LIN {X 0,Y 525.784,Z 203.51,A -85,B 0,C 180,E1 -4784.972,E2 -4784.972} C_VEL
LIN {X 0,Y 524.23,Z 193.259,A -85,B 0,C 180,E1 -4785.175,E2 -4785.175} C_VEL
LIN {X 0,Y 524.605,Z 174.888,A -85,B 0,C 180,E1 -4787.978,E2 -4787.978} C_VEL
LIN {X 0,Y 525.075,Z 155.446,A -85,B 0,C 180,E1 -4790.98,E2 -4790.98} C_VEL
LIN {X 0,Y 525.35,Z 141.019,A -85,B 0,C 180,E1 -4793.244,E2 -4793.244} C_VEL
LIN {X 0,Y 523.931,Z 133.223,A -85,B 0,C 180,E1 -4794.572,E2 -4794.572} C_VEL
LIN {X 0,Y 523.922,Z 133.227,A -85,B 0,C 180,E1 -4797.706,E2 -4797.706} C_VEL
LIN {X 0,Y 523.948,Z 133.217,A -85,B 0,C 180,E1 -4800.645,E2 -4800.645} C_VEL
LIN {X 0,Y 523.93,Z 133.224,A -85,B 0,C 180,E1 -4803.729,E2 -4803.729} C_VEL
LIN {X 0,Y 523.902,Z 133.221,A -85,B 0,C 180,E1 -4806.4,E2 -4806.4} C_VEL
LIN {X 0,Y 523.916,Z 133.222,A -85,B 0,C 180,E1 -4809.086,E2 -4809.086} C_VEL
LIN {X 0,Y 523.903,Z 133.221,A -85,B 0,C 180,E1 -4812.124,E2 -4812.124} C_VEL
LIN {X 0,Y 523.938,Z 133.225,A -85,B 0,C 180,E1 -4815.311,E2 -4815.311} C_VEL
LIN {X 0,Y 523.925,Z 133.22,A -85,B 0,C 180,E1 -4818.694,E2 -4818.694} C_VEL
LIN {X 0,Y 523.916,Z 133.219,A -85,B 0,C 180,E1 -4821.898,E2 -4821.898} C_VEL
LIN {X 0,Y 523.922,Z 133.225,A -85,B 0,C 180,E1 -4824.912,E2 -4824.912} C_VEL
LIN {X 0,Y 523.935,Z 133.217,A -85,B 0,C 180,E1 -4827.681,E2 -4827.681} C_VEL
LIN {X 0,Y 523.936,Z 133.221,A -85,B 0,C 180,E1 -4830.681,E2 -4830.681} C_VEL
LIN {X 0,Y 523.908,Z 133.22,A -85,B 0,C 180,E1 -4833.724,E2 -4833.724} C_VEL
LIN {X 0,Y 523.903,Z 133.222,A -85,B 0,C 180,E1 -4836.269,E2 -4836.269} C_VEL
LIN {X 0,Y 523.929,Z 133.226,A -85,B 0,C 180,E1 -4838.765,E2 -4838.765} C_VEL
LIN {X 0,Y 523.931,Z 133.219,A -85,B 0,C 180,E1 -4841.219,E2 -4841.219} C_VEL
LIN {X 0,Y 523.915,Z 133.225,A -85,B 0,C 180,E1 -4844.437,E2 -4844.437} C_VEL
LIN {X 0,Y 523.955,Z 133.214,A -85,B 0,C 180,E1 -4847.607,E2 -4847.607} C_VEL
LIN {X 0,Y 523.933,Z 133.219,A -85,B 0,C 180,E1 -4849.957,E2 -4849.957} C_VEL
LIN {X 0,Y 523.997,Z 133.209,A -85,B 0,C 180,E1 -4853.066,E2 -4853.066} C_VEL
LIN {X 0,Y 523.95,Z 133.214,A -85,B 0,C 180,E1 -4855.383,E2 -4855.383} C_VEL
LIN {X 0,Y 524.107,Z 133.196,A -85,B 0,C 180,E1 -4857.694,E2 -4857.694} C_VEL
LIN {X 0,Y 524.1,Z 133.201,A -85,B 0,C 180,E1 -4859.999,E2 -4859.999} C_VEL
LIN {X 0,Y 524.107,Z 133.202,A -85,B 0,C 180,E1 -4862.305,E2 -4862.305} C_VEL
LIN {X 0,Y 524.004,Z 133.216,A -85,B 0,C 180,E1 -4866.159,E2 -4866.159} C_VEL
LIN {X 0,Y 523.948,Z 133.215,A -85,B 0,C 180,E1 -4869.262,E2 -4869.262} C_VEL
LIN {X 0,Y 523.949,Z 133.217,A -85,B 0,C 180,E1 -4872.392,E2 -4872.392} C_VEL
LIN {X 0,Y 523.986,Z 133.21,A -85,B 0,C 180,E1 -4875.047,E2 -4875.047} C_VEL
LIN {X 0,Y 523.912,Z 133.226,A -85,B 0,C 180,E1 -4877.97,E2 -4877.97} C_VEL
LIN {X 0,Y 523.917,Z 133.219,A -85,B 0,C 180,E1 -4880.411,E2 -4880.411} C_VEL
LIN {X 0,Y 523.887,Z 133.223,A -85,B 0,C 180,E1 -4882.894,E2 -4882.894} C_VEL
LIN {X 0,Y 523.899,Z 133.227,A -85,B 0,C 180,E1 -4885.421,E2 -4885.421} C_VEL
LIN {X 0,Y 523.896,Z 133.224,A -85,B 0,C 180,E1 -4888.002,E2 -4888.002} C_VEL
LIN {X 0,Y 523.901,Z 133.222,A -85,B 0,C 180,E1 -4890.846,E2 -4890.846} C_VEL
LIN {X 0,Y 523.925,Z 133.222,A -85,B 0,C 180,E1 -4893.728,E2 -4893.728} C_VEL
LIN {X 0,Y 523.885,Z 133.222,A -85,B 0,C 180,E1 -4896.398,E2 -4896.398} C_VEL
LIN {X 0,Y 523.907,Z 133.226,A -85,B 0,C 180,E1 -4899.085,E2 -4899.085} C_VEL
LIN {X 0,Y 523.889,Z 133.222,A -85,B 0,C 180,E1 -4902.124,E2 -4902.124} C_VEL
LIN {X 0,Y 523.93,Z 133.223,A -85,B 0,C 180,E1 -4905.31,E2 -4905.31} C_VEL
LIN {X 0,Y 523.874,Z 133.228,A -85,B 0,C 180,E1 -4906.873,E2 -4906.873} C_VEL
LIN {X 0,Y 523.187,Z 133.313,A -85,B 0,C 180,E1 -4907.514,E2 -4907.514} C_VEL
LIN {X 0,Y 520.323,Z 133.669,A -85,B 0,C 180,E1 -4908.556,E2 -4908.556} C_VEL
LIN {X 0,Y 517.929,Z 133.968,A -85,B 0,C 180,E1 -4909.395,E2 -4909.395} C_VEL
LIN {X 0,Y 516.923,Z 134.09,A -85,B 0,C 180,E1 -4910.043,E2 -4910.043} C_VEL
LIN {X 0,Y 516.853,Z 134.099,A -85,B 0,C 180,E1 -4910.262,E2 -4910.262} C_VEL
LIN {X 0,Y 516.844,Z 134.104,A -85,B 0,C 180,E1 -4913.251,E2 -4913.251} C_VEL
LIN {X 0,Y 516.873,Z 134.096,A -85,B 0,C 180,E1 -4916.118,E2 -4916.118} C_VEL
LIN {X 0,Y 516.872,Z 134.103,A -85,B 0,C 180,E1 -4918.938,E2 -4918.938} C_VEL
LIN {X 0,Y 516.838,Z 134.101,A -85,B 0,C 180,E1 -4921.58,E2 -4921.58} C_VEL
LIN {X 0,Y 516.863,Z 134.1,A -85,B 0,C 180,E1 -4924.207,E2 -4924.207} C_VEL
LIN {X 0,Y 516.834,Z 134.107,A -85,B 0,C 180,E1 -4926.774,E2 -4926.774} C_VEL
LIN {X 0,Y 516.9,Z 134.093,A -85,B 0,C 180,E1 -4929.741,E2 -4929.741} C_VEL
LIN {X 0,Y 516.857,Z 134.105,A -85,B 0,C 180,E1 -4932.593,E2 -4932.593} C_VEL
LIN {X 0,Y 516.924,Z 134.091,A -85,B 0,C 180,E1 -4935.029,E2 -4935.029} C_VEL
LIN {X 0,Y 516.918,Z 134.098,A -85,B 0,C 180,E1 -4938.232,E2 -4938.232} C_VEL
LIN {X 0,Y 516.911,Z 134.091,A -85,B 0,C 180,E1 -4941.399,E2 -4941.399} C_VEL
LIN {X 0,Y 516.973,Z 134.088,A -85,B 0,C 180,E1 -4944.539,E2 -4944.539} C_VEL
LIN {X 0,Y 517.065,Z 134.077,A -85,B 0,C 180,E1 -4947.663,E2 -4947.663} C_VEL
LIN {X 0,Y 517.057,Z 134.082,A -85,B 0,C 180,E1 -4950,E2 -4950} C_VEL
LIN {X 0,Y 517.019,Z 134.112,A -85,B 0,C 180,E1 -4952.093,E2 -4952.093} C_VEL
LIN {X 0,Y 517.465,Z 141.303,A -85,B 0,C 180,E1 -4953.504,E2 -4953.504} C_VEL
LIN {X 0,Y 517.243,Z 157.8,A -85,B 0,C 180,E1 -4956.681,E2 -4956.681} C_VEL
LIN {X 0,Y 519.137,Z 168.241,A -85,B 0,C 180,E1 -4956.901,E2 -4956.901} C_VEL
LIN {X 0,Y 518.63,Z 265.183,A -85,B 0,C 180,E1 -4958.273,E2 -4958.273} C_VEL
LIN {X 0,Y 518.353,Z 278.542,A -85,B 0,C 180,E1 -4958.626,E2 -4958.626} C_VEL
LIN {X 0,Y 518.211,Z 291.011,A -85,B 0,C 180,E1 -4959.12,E2 -4959.12} C_VEL
LIN {X 0,Y 517.946,Z 302.998,A -85,B 0,C 180,E1 -4959.765,E2 -4959.765} C_VEL
LIN {X 0,Y 517.637,Z 314.493,A -85,B 0,C 180,E1 -4960.561,E2 -4960.561} C_VEL
LIN {X 0,Y 517.37,Z 324.842,A -85,B 0,C 180,E1 -4961.459,E2 -4961.459} C_VEL
LIN {X 0,Y 517.072,Z 333.267,A -85,B 0,C 180,E1 -4962.353,E2 -4962.353} C_VEL
LIN {X 0,Y 516.809,Z 342.529,A -85,B 0,C 180,E1 -4963.567,E2 -4963.567} C_VEL
LIN {X 0,Y 516.59,Z 349.95,A -85,B 0,C 180,E1 -4964.779,E2 -4964.779} C_VEL
LIN {X 0,Y 516.491,Z 354.945,A -85,B 0,C 180,E1 -4965.792,E2 -4965.792} C_VEL
LIN {X 0,Y 516.368,Z 359.797,A -85,B 0,C 180,E1 -4967.015,E2 -4967.015} C_VEL
LIN {X 0,Y 516.301,Z 363.48,A -85,B 0,C 180,E1 -4968.245,E2 -4968.245} C_VEL
LIN {X 0,Y 516.228,Z 365.322,A -85,B 0,C 180,E1 -4969.071,E2 -4969.071} C_VEL
LIN {X 0,Y 516.221,Z 366.922,A -85,B 0,C 180,E1 -4970.054,E2 -4970.054} C_VEL
LIN {X 0,Y 516.19,Z 368.129,A -85,B 0,C 180,E1 -4971.568,E2 -4971.568} C_VEL
LIN {X 0,Y 516.194,Z 368.154,A -85,B 0,C 180,E1 -4972.409,E2 -4972.409} C_VEL
LIN {X 0,Y 516.191,Z 367.747,A -85,B 0,C 180,E1 -4973.256,E2 -4973.256} C_VEL
LIN {X 0,Y 516.211,Z 366.705,A -85,B 0,C 180,E1 -4974.194,E2 -4974.194} C_VEL
LIN {X 0,Y 516.231,Z 365.437,A -85,B 0,C 180,E1 -4974.963,E2 -4974.963} C_VEL
LIN {X 0,Y 516.341,Z 362.91,A -85,B 0,C 180,E1 -4976.062,E2 -4976.062} C_VEL
LIN {X 0,Y 516.419,Z 358.059,A -85,B 0,C 180,E1 -4977.562,E2 -4977.562} C_VEL
LIN {X 0,Y 516.522,Z 352.207,A -85,B 0,C 180,E1 -4978.883,E2 -4978.883} C_VEL
LIN {X 0,Y 516.722,Z 344.637,A -85,B 0,C 180,E1 -4980.215,E2 -4980.215} C_VEL
LIN {X 0,Y 516.947,Z 336.655,A -85,B 0,C 180,E1 -4981.333,E2 -4981.333} C_VEL
LIN {X 0,Y 517.233,Z 327.241,A -85,B 0,C 180,E1 -4982.397,E2 -4982.397} C_VEL
LIN {X 0,Y 517.536,Z 316.641,A -85,B 0,C 180,E1 -4983.366,E2 -4983.366} C_VEL
LIN {X 0,Y 517.872,Z 306.251,A -85,B 0,C 180,E1 -4984.126,E2 -4984.126} C_VEL
LIN {X 0,Y 518.18,Z 294.832,A -85,B 0,C 180,E1 -4984.784,E2 -4984.784} C_VEL
LIN {X 0,Y 518.398,Z 281.579,A -85,B 0,C 180,E1 -4985.361,E2 -4985.361} C_VEL
LIN {X 0,Y 518.578,Z 268.396,A -85,B 0,C 180,E1 -4985.749,E2 -4985.749} C_VEL
LIN {X 0,Y 518.706,Z 250.944,A -85,B 0,C 180,E1 -4986.038,E2 -4986.038} C_VEL
LIN {X 0,Y 519.017,Z 166.958,A -85,B 0,C 180,E1 -4987.213,E2 -4987.213} C_VEL
LIN {X 0,Y 517.321,Z 157.839,A -85,B 0,C 180,E1 -4987.414,E2 -4987.414} C_VEL
LIN {X 0,Y 517.561,Z 140.56,A -85,B 0,C 180,E1 -4990.677,E2 -4990.677} C_VEL
LIN {X 0,Y 516.974,Z 134.465,A -85,B 0,C 180,E1 -4991.86,E2 -4991.86} C_VEL
LIN {X 0,Y 516.92,Z 134.099,A -85,B 0,C 180,E1 -4991.974,E2 -4991.974} C_VEL
LIN {X 0,Y 516.919,Z 134.094,A -85,B 0,C 180,E1 -4995.011,E2 -4995.011} C_VEL
LIN {X 0,Y 516.92,Z 134.095,A -85,B 0,C 180,E1 -4998.398,E2 -4998.398} C_VEL
LIN {X 0,Y 516.884,Z 134.099,A -85,B 0,C 180,E1 -5001.285,E2 -5001.285} C_VEL
LIN {X 0,Y 516.868,Z 134.1,A -85,B 0,C 180,E1 -5004.22,E2 -5004.22} C_VEL
LIN {X 0,Y 516.892,Z 134.097,A -85,B 0,C 180,E1 -5007.054,E2 -5007.054} C_VEL
LIN {X 0,Y 516.89,Z 134.098,A -85,B 0,C 180,E1 -5009.797,E2 -5009.797} C_VEL
LIN {X 0,Y 516.925,Z 134.091,A -85,B 0,C 180,E1 -5012.468,E2 -5012.468} C_VEL
LIN {X 0,Y 516.908,Z 134.099,A -85,B 0,C 180,E1 -5015.073,E2 -5015.073} C_VEL
LIN {X 0,Y 516.885,Z 134.097,A -85,B 0,C 180,E1 -5018.463,E2 -5018.463} C_VEL
LIN {X 0,Y 516.893,Z 134.101,A -85,B 0,C 180,E1 -5020.955,E2 -5020.955} C_VEL
LIN {X 0,Y 516.898,Z 134.097,A -85,B 0,C 180,E1 -5023.41,E2 -5023.41} C_VEL
LIN {X 0,Y 516.888,Z 134.094,A -85,B 0,C 180,E1 -5025.834,E2 -5025.834} C_VEL
LIN {X 0,Y 516.952,Z 134.092,A -85,B 0,C 180,E1 -5029.029,E2 -5029.029} C_VEL
LIN {X 0,Y 516.964,Z 134.085,A -85,B 0,C 180,E1 -5032.187,E2 -5032.187} C_VEL
LIN {X 0,Y 517.025,Z 134.085,A -85,B 0,C 180,E1 -5034.541,E2 -5034.541} C_VEL
LIN {X 0,Y 517.082,Z 134.069,A -85,B 0,C 180,E1 -5037.664,E2 -5037.664} C_VEL
LIN {X 0,Y 517.091,Z 134.069,A -85,B 0,C 180,E1 -5040.779,E2 -5040.779} C_VEL
LIN {X 0,Y 516.95,Z 134.086,A -85,B 0,C 180,E1 -5043.118,E2 -5043.118} C_VEL
LIN {X 0,Y 516.974,Z 134.087,A -85,B 0,C 180,E1 -5046.244,E2 -5046.244} C_VEL
LIN {X 0,Y 516.939,Z 134.088,A -85,B 0,C 180,E1 -5049.39,E2 -5049.39} C_VEL
LIN {X 0,Y 516.956,Z 134.087,A -85,B 0,C 180,E1 -5051.807,E2 -5051.807} C_VEL
LIN {X 0,Y 516.946,Z 134.087,A -85,B 0,C 180,E1 -5055.146,E2 -5055.146} C_VEL
LIN {X 0,Y 516.877,Z 134.1,A -85,B 0,C 180,E1 -5058.225,E2 -5058.225} C_VEL
LIN {X 0,Y 516.882,Z 134.094,A -85,B 0,C 180,E1 -5060.703,E2 -5060.703} C_VEL
LIN {X 0,Y 516.842,Z 134.102,A -85,B 0,C 180,E1 -5063.225,E2 -5063.225} C_VEL
LIN {X 0,Y 516.881,Z 134.094,A -85,B 0,C 180,E1 -5066.182,E2 -5066.182} C_VEL
LIN {X 0,Y 516.831,Z 134.102,A -85,B 0,C 180,E1 -5068.421,E2 -5068.421} C_VEL
LIN {X 0,Y 516.85,Z 134.102,A -85,B 0,C 180,E1 -5071.113,E2 -5071.113} C_VEL
LIN {X 0,Y 516.87,Z 134.096,A -85,B 0,C 180,E1 -5073.959,E2 -5073.959} C_VEL
LIN {X 0,Y 516.801,Z 134.109,A -85,B 0,C 180,E1 -5076.753,E2 -5076.753} C_VEL
LIN {X 0,Y 516.826,Z 134.105,A -85,B 0,C 180,E1 -5079.727,E2 -5079.727} C_VEL
LIN {X 0,Y 516.843,Z 134.108,A -85,B 0,C 180,E1 -5082.836,E2 -5082.836} C_VEL
LIN {X 0,Y 516.898,Z 134.103,A -85,B 0,C 180,E1 -5085.007,E2 -5085.007} C_VEL
LIN {X 0,Y 516.851,Z 134.105,A -85,B 0,C 180,E1 -5088.407,E2 -5088.407} C_VEL
LIN {X 0,Y 516.876,Z 134.099,A -85,B 0,C 180,E1 -5091.284,E2 -5091.284} C_VEL
LIN {X 0,Y 516.858,Z 134.101,A -85,B 0,C 180,E1 -5094.219,E2 -5094.219} C_VEL
LIN {X 0,Y 516.883,Z 134.099,A -85,B 0,C 180,E1 -5097.052,E2 -5097.052} C_VEL
LIN {X 0,Y 516.869,Z 134.1,A -85,B 0,C 180,E1 -5099.795,E2 -5099.795} C_VEL
LIN {X 0,Y 516.877,Z 134.104,A -85,B 0,C 180,E1 -5102.464,E2 -5102.464} C_VEL
LIN {X 0,Y 516.919,Z 134.232,A -85,B 0,C 180,E1 -5105.385,E2 -5105.385} C_VEL
LIN {X 0,Y 518.398,Z 142.946,A -85,B 0,C 180,E1 -5106.849,E2 -5106.849} C_VEL
LIN {X 0,Y 517.904,Z 161.656,A -85,B 0,C 180,E1 -5109.793,E2 -5109.793} C_VEL
LIN {X 0,Y 517.514,Z 178.694,A -85,B 0,C 180,E1 -5112.438,E2 -5112.438} C_VEL
LIN {X 0,Y 517.204,Z 192.95,A -85,B 0,C 180,E1 -5114.63,E2 -5114.63} C_VEL
LIN {X 0,Y 519.009,Z 206.524,A -85,B 0,C 180,E1 -5114.875,E2 -5114.875} C_VEL
LIN {X 0,Y 518.601,Z 300.988,A -85,B 0,C 180,E1 -5116.206,E2 -5116.206} C_VEL
LIN {X 0,Y 518.369,Z 314.405,A -85,B 0,C 180,E1 -5116.55,E2 -5116.55} C_VEL
LIN {X 0,Y 518.088,Z 326.647,A -85,B 0,C 180,E1 -5117.016,E2 -5117.016} C_VEL
LIN {X 0,Y 517.783,Z 338.229,A -85,B 0,C 180,E1 -5117.61,E2 -5117.61} C_VEL
LIN {X 0,Y 517.52,Z 349.342,A -85,B 0,C 180,E1 -5118.346,E2 -5118.346} C_VEL
LIN {X 0,Y 517.231,Z 360.049,A -85,B 0,C 180,E1 -5119.232,E2 -5119.232} C_VEL
LIN {X 0,Y 516.907,Z 369.696,A -85,B 0,C 180,E1 -5120.215,E2 -5120.215} C_VEL
LIN {X 0,Y 516.693,Z 377.606,A -85,B 0,C 180,E1 -5121.198,E2 -5121.198} C_VEL
LIN {X 0,Y 516.523,Z 385.334,A -85,B 0,C 180,E1 -5122.377,E2 -5122.377} C_VEL
LIN {X 0,Y 516.376,Z 392.455,A -85,B 0,C 180,E1 -5123.749,E2 -5123.749} C_VEL
LIN {X 0,Y 516.312,Z 397.195,A -85,B 0,C 180,E1 -5124.924,E2 -5124.924} C_VEL
LIN {X 0,Y 516.352,Z 400.82,A -85,B 0,C 180,E1 -5126.098,E2 -5126.098} C_VEL
LIN {X 0,Y 516.283,Z 402.686,A -85,B 0,C 180,E1 -5126.879,E2 -5126.879} C_VEL
LIN {X 0,Y 516.262,Z 404.087,A -85,B 0,C 180,E1 -5127.66,E2 -5127.66} C_VEL
LIN {X 0,Y 516.166,Z 405.696,A -85,B 0,C 180,E1 -5129.22,E2 -5129.22} C_VEL
LIN {X 0,Y 516.164,Z 405.915,A -85,B 0,C 180,E1 -5130,E2 -5130} C_VEL
LIN {X 0,Y 516.192,Z 405.094,A -85,B 0,C 180,E1 -5131.561,E2 -5131.561} C_VEL
LIN {X 0,Y 516.262,Z 404.101,A -85,B 0,C 180,E1 -5132.341,E2 -5132.341} C_VEL
LIN {X 0,Y 516.283,Z 402.704,A -85,B 0,C 180,E1 -5133.122,E2 -5133.122} C_VEL
LIN {X 0,Y 516.31,Z 399.764,A -85,B 0,C 180,E1 -5134.294,E2 -5134.294} C_VEL
LIN {X 0,Y 516.367,Z 395.783,A -85,B 0,C 180,E1 -5135.467,E2 -5135.467} C_VEL
LIN {X 0,Y 516.413,Z 390.609,A -85,B 0,C 180,E1 -5136.653,E2 -5136.653} C_VEL
LIN {X 0,Y 516.545,Z 384.205,A -85,B 0,C 180,E1 -5137.82,E2 -5137.82} C_VEL
LIN {X 0,Y 516.749,Z 376.158,A -85,B 0,C 180,E1 -5138.998,E2 -5138.998} C_VEL
LIN {X 0,Y 516.943,Z 367.956,A -85,B 0,C 180,E1 -5139.982,E2 -5139.982} C_VEL
LIN {X 0,Y 517.29,Z 357.958,A -85,B 0,C 180,E1 -5140.965,E2 -5140.965} C_VEL
LIN {X 0,Y 517.592,Z 348.09,A -85,B 0,C 180,E1 -5141.752,E2 -5141.752} C_VEL
LIN {X 0,Y 517.843,Z 336.945,A -85,B 0,C 180,E1 -5142.466,E2 -5142.466} C_VEL
LIN {X 0,Y 518.126,Z 324.456,A -85,B 0,C 180,E1 -5143.083,E2 -5143.083} C_VEL
LIN {X 0,Y 518.424,Z 311.314,A -85,B 0,C 180,E1 -5143.549,E2 -5143.549} C_VEL
LIN {X 0,Y 518.668,Z 298.153,A -85,B 0,C 180,E1 -5143.842,E2 -5143.842} C_VEL
LIN {X 0,Y 518.977,Z 204.563,A -85,B 0,C 180,E1 -5145.155,E2 -5145.155} C_VEL
LIN {X 0,Y 517.23,Z 192.979,A -85,B 0,C 180,E1 -5145.39,E2 -5145.39} C_VEL
LIN {X 0,Y 517.637,Z 174.838,A -85,B 0,C 180,E1 -5148.197,E2 -5148.197} C_VEL
LIN {X 0,Y 518.13,Z 155.204,A -85,B 0,C 180,E1 -5151.275,E2 -5151.275} C_VEL
LIN {X 0,Y 518.395,Z 142.093,A -85,B 0,C 180,E1 -5153.363,E2 -5153.363} C_VEL
LIN {X 0,Y 516.89,Z 134.1,A -85,B 0,C 180,E1 -5154.742,E2 -5154.742} C_VEL
LIN {X 0,Y 516.868,Z 134.104,A -85,B 0,C 180,E1 -5157.892,E2 -5157.892} C_VEL
LIN {X 0,Y 516.871,Z 134.101,A -85,B 0,C 180,E1 -5160.205,E2 -5160.205} C_VEL
LIN {X 0,Y 516.884,Z 134.096,A -85,B 0,C 180,E1 -5162.948,E2 -5162.948} C_VEL
LIN {X 0,Y 516.87,Z 134.102,A -85,B 0,C 180,E1 -5165.781,E2 -5165.781} C_VEL
LIN {X 0,Y 516.88,Z 134.096,A -85,B 0,C 180,E1 -5168.716,E2 -5168.716} C_VEL
LIN {X 0,Y 516.854,Z 134.102,A -85,B 0,C 180,E1 -5171.781,E2 -5171.781} C_VEL
LIN {X 0,Y 516.901,Z 134.097,A -85,B 0,C 180,E1 -5175.007,E2 -5175.007} C_VEL
LIN {X 0,Y 516.86,Z 134.098,A -85,B 0,C 180,E1 -5178.406,E2 -5178.406} C_VEL
LIN {X 0,Y 516.88,Z 134.102,A -85,B 0,C 180,E1 -5181.283,E2 -5181.283} C_VEL
LIN {X 0,Y 516.871,Z 134.096,A -85,B 0,C 180,E1 -5184.219,E2 -5184.219} C_VEL
LIN {X 0,Y 516.884,Z 134.103,A -85,B 0,C 180,E1 -5187.052,E2 -5187.052} C_VEL
LIN {X 0,Y 516.85,Z 134.099,A -85,B 0,C 180,E1 -5189.793,E2 -5189.793} C_VEL
LIN {X 0,Y 516.88,Z 134.098,A -85,B 0,C 180,E1 -5192.464,E2 -5192.464} C_VEL
LIN {X 0,Y 516.849,Z 134.104,A -85,B 0,C 180,E1 -5195.068,E2 -5195.068} C_VEL
LIN {X 0,Y 516.875,Z 134.096,A -85,B 0,C 180,E1 -5197.621,E2 -5197.621} C_VEL
LIN {X 0,Y 516.92,Z 134.092,A -85,B 0,C 180,E1 -5200.129,E2 -5200.129} C_VEL
LIN {X 0,Y 516.87,Z 134.105,A -85,B 0,C 180,E1 -5202.594,E2 -5202.594} C_VEL
LIN {X 0,Y 516.936,Z 134.091,A -85,B 0,C 180,E1 -5205.029,E2 -5205.029} C_VEL
LIN {X 0,Y 516.973,Z 134.088,A -85,B 0,C 180,E1 -5208.233,E2 -5208.233} C_VEL
LIN {X 0,Y 516.931,Z 134.089,A -85,B 0,C 180,E1 -5211.398,E2 -5211.398} C_VEL
LIN {X 0,Y 516.985,Z 134.088,A -85,B 0,C 180,E1 -5214.539,E2 -5214.539} C_VEL
LIN {X 0,Y 517.077,Z 134.072,A -85,B 0,C 180,E1 -5217.662,E2 -5217.662} C_VEL
LIN {X 0,Y 517.069,Z 134.077,A -85,B 0,C 180,E1 -5219.999,E2 -5219.999} C_VEL
LIN {X 0,Y 517.077,Z 134.077,A -85,B 0,C 180,E1 -5222.336,E2 -5222.336} C_VEL
LIN {X 0,Y 516.971,Z 134.09,A -85,B 0,C 180,E1 -5226.243,E2 -5226.243} C_VEL
LIN {X 0,Y 516.91,Z 134.093,A -85,B 0,C 180,E1 -5229.389,E2 -5229.389} C_VEL
LIN {X 0,Y 516.901,Z 134.094,A -85,B 0,C 180,E1 -5232.564,E2 -5232.564} C_VEL
LIN {X 0,Y 516.938,Z 134.089,A -85,B 0,C 180,E1 -5235.141,E2 -5235.141} C_VEL
LIN {X 0,Y 516.872,Z 134.099,A -85,B 0,C 180,E1 -5238.223,E2 -5238.223} C_VEL
LIN {X 0,Y 516.872,Z 134.096,A -85,B 0,C 180,E1 -5240.702,E2 -5240.702} C_VEL
LIN {X 0,Y 516.842,Z 134.103,A -85,B 0,C 180,E1 -5243.224,E2 -5243.224} C_VEL
LIN {X 0,Y 516.879,Z 134.097,A -85,B 0,C 180,E1 -5246.18,E2 -5246.18} C_VEL
LIN {X 0,Y 516.889,Z 134.1,A -85,B 0,C 180,E1 -5249.306,E2 -5249.306} C_VEL
LIN {X 0,Y 516.891,Z 134.094,A -85,B 0,C 180,E1 -5252.542,E2 -5252.542} C_VEL
LIN {X 0,Y 516.853,Z 134.107,A -85,B 0,C 180,E1 -5255.327,E2 -5255.327} C_VEL
LIN {X 0,Y 516.874,Z 134.097,A -85,B 0,C 180,E1 -5257.941,E2 -5257.941} C_VEL
LIN {X 0,Y 516.844,Z 134.102,A -85,B 0,C 180,E1 -5260.744,E2 -5260.744} C_VEL
LIN {X 0,Y 516.877,Z 134.096,A -85,B 0,C 180,E1 -5263.903,E2 -5263.903} C_VEL
LIN {X 0,Y 516.83,Z 134.105,A -85,B 0,C 180,E1 -5266.873,E2 -5266.873} C_VEL
LIN {X 0,Y 516.854,Z 134.1,A -85,B 0,C 180,E1 -5269.592,E2 -5269.592} C_VEL
LIN {X 0,Y 516.853,Z 134.099,A -85,B 0,C 180,E1 -5270.262,E2 -5270.262} C_VEL
LIN {X 0,Y 516.215,Z 134.186,A -85,B 0,C 180,E1 -5270.912,E2 -5270.912} C_VEL
LIN {X 0,Y 513.369,Z 134.538,A -85,B 0,C 180,E1 -5271.968,E2 -5271.968} C_VEL
LIN {X 0,Y 510.939,Z 134.842,A -85,B 0,C 180,E1 -5272.818,E2 -5272.818} C_VEL
LIN {X 0,Y 509.885,Z 134.969,A -85,B 0,C 180,E1 -5273.475,E2 -5273.475} C_VEL
LIN {X 0,Y 509.795,Z 134.978,A -85,B 0,C 180,E1 -5273.697,E2 -5273.697} C_VEL
LIN {X 0,Y 509.833,Z 134.977,A -85,B 0,C 180,E1 -5276.537,E2 -5276.537} C_VEL
LIN {X 0,Y 509.815,Z 134.977,A -85,B 0,C 180,E1 -5279.332,E2 -5279.332} C_VEL
LIN {X 0,Y 509.823,Z 134.975,A -85,B 0,C 180,E1 -5282.05,E2 -5282.05} C_VEL
LIN {X 0,Y 509.794,Z 134.986,A -85,B 0,C 180,E1 -5284.699,E2 -5284.699} C_VEL
LIN {X 0,Y 509.817,Z 134.975,A -85,B 0,C 180,E1 -5287.458,E2 -5287.458} C_VEL
LIN {X 0,Y 509.882,Z 134.968,A -85,B 0,C 180,E1 -5289.843,E2 -5289.843} C_VEL
LIN {X 0,Y 509.839,Z 134.979,A -85,B 0,C 180,E1 -5292.346,E2 -5292.346} C_VEL
LIN {X 0,Y 509.877,Z 134.971,A -85,B 0,C 180,E1 -5294.817,E2 -5294.817} C_VEL
LIN {X 0,Y 509.881,Z 134.973,A -85,B 0,C 180,E1 -5298.13,E2 -5298.13} C_VEL
LIN {X 0,Y 509.864,Z 134.969,A -85,B 0,C 180,E1 -5301.279,E2 -5301.279} C_VEL
LIN {X 0,Y 509.908,Z 134.966,A -85,B 0,C 180,E1 -5303.669,E2 -5303.669} C_VEL
LIN {X 0,Y 509.877,Z 134.97,A -85,B 0,C 180,E1 -5306.839,E2 -5306.839} C_VEL
LIN {X 0,Y 509.915,Z 134.97,A -85,B 0,C 180,E1 -5308.42,E2 -5308.42} C_VEL
LIN {X 0,Y 510.026,Z 134.958,A -85,B 0,C 180,E1 -5310,E2 -5310} C_VEL
LIN {X 0,Y 509.974,Z 135.051,A -85,B 0,C 180,E1 -5311.974,E2 -5311.974} C_VEL
LIN {X 0,Y 510.488,Z 140.984,A -85,B 0,C 180,E1 -5313.157,E2 -5313.157} C_VEL
LIN {X 0,Y 510.294,Z 157.282,A -85,B 0,C 180,E1 -5316.326,E2 -5316.326} C_VEL
LIN {X 0,Y 510.269,Z 158.053,A -85,B 0,C 180,E1 -5316.475,E2 -5316.475} C_VEL
LIN {X 0,Y 512.292,Z 168.671,A -85,B 0,C 180,E1 -5316.696,E2 -5316.696} C_VEL
LIN {X 0,Y 511.734,Z 264.788,A -85,B 0,C 180,E1 -5318.071,E2 -5318.071} C_VEL
LIN {X 0,Y 511.506,Z 277.724,A -85,B 0,C 180,E1 -5318.409,E2 -5318.409} C_VEL
LIN {X 0,Y 511.313,Z 290.184,A -85,B 0,C 180,E1 -5318.895,E2 -5318.895} C_VEL
LIN {X 0,Y 511.097,Z 301.642,A -85,B 0,C 180,E1 -5319.498,E2 -5319.498} C_VEL
LIN {X 0,Y 510.763,Z 312.167,A -85,B 0,C 180,E1 -5320.204,E2 -5320.204} C_VEL
LIN {X 0,Y 510.416,Z 322.987,A -85,B 0,C 180,E1 -5321.114,E2 -5321.114} C_VEL
LIN {X 0,Y 510.1,Z 332.554,A -85,B 0,C 180,E1 -5322.108,E2 -5322.108} C_VEL
LIN {X 0,Y 509.827,Z 340.724,A -85,B 0,C 180,E1 -5323.147,E2 -5323.147} C_VEL
LIN {X 0,Y 509.615,Z 348.497,A -85,B 0,C 180,E1 -5324.373,E2 -5324.373} C_VEL
LIN {X 0,Y 509.43,Z 354.75,A -85,B 0,C 180,E1 -5325.606,E2 -5325.606} C_VEL
LIN {X 0,Y 509.307,Z 359.693,A -85,B 0,C 180,E1 -5326.845,E2 -5326.845} C_VEL
LIN {X 0,Y 509.251,Z 362.637,A -85,B 0,C 180,E1 -5327.781,E2 -5327.781} C_VEL
LIN {X 0,Y 509.148,Z 366.156,A -85,B 0,C 180,E1 -5329.347,E2 -5329.347} C_VEL
LIN {X 0,Y 509.131,Z 367.385,A -85,B 0,C 180,E1 -5330.188,E2 -5330.188} C_VEL
LIN {X 0,Y 509.085,Z 368.132,A -85,B 0,C 180,E1 -5331.035,E2 -5331.035} C_VEL
LIN {X 0,Y 509.103,Z 368.426,A -85,B 0,C 180,E1 -5332.347,E2 -5332.347} C_VEL
LIN {X 0,Y 509.108,Z 367.7,A -85,B 0,C 180,E1 -5333.599,E2 -5333.599} C_VEL
LIN {X 0,Y 509.118,Z 366.627,A -85,B 0,C 180,E1 -5334.464,E2 -5334.464} C_VEL
LIN {X 0,Y 509.22,Z 364.073,A -85,B 0,C 180,E1 -5335.769,E2 -5335.769} C_VEL
LIN {X 0,Y 509.332,Z 360.285,A -85,B 0,C 180,E1 -5337.087,E2 -5337.087} C_VEL
LIN {X 0,Y 509.403,Z 355.071,A -85,B 0,C 180,E1 -5338.423,E2 -5338.423} C_VEL
LIN {X 0,Y 509.603,Z 348.267,A -85,B 0,C 180,E1 -5339.767,E2 -5339.767} C_VEL
LIN {X 0,Y 509.794,Z 341.287,A -85,B 0,C 180,E1 -5340.87,E2 -5340.87} C_VEL
LIN {X 0,Y 510.119,Z 332.153,A -85,B 0,C 180,E1 -5342.034,E2 -5342.034} C_VEL
LIN {X 0,Y 510.465,Z 321.822,A -85,B 0,C 180,E1 -5343.092,E2 -5343.092} C_VEL
LIN {X 0,Y 510.788,Z 310.918,A -85,B 0,C 180,E1 -5343.984,E2 -5343.984} C_VEL
LIN {X 0,Y 511.123,Z 299.044,A -85,B 0,C 180,E1 -5344.746,E2 -5344.746} C_VEL
LIN {X 0,Y 511.442,Z 286.74,A -85,B 0,C 180,E1 -5345.35,E2 -5345.35} C_VEL
LIN {X 0,Y 511.646,Z 274.423,A -85,B 0,C 180,E1 -5345.785,E2 -5345.785} C_VEL
LIN {X 0,Y 511.778,Z 261.825,A -85,B 0,C 180,E1 -5346.072,E2 -5346.072} C_VEL
LIN {X 0,Y 512.205,Z 167.918,A -85,B 0,C 180,E1 -5347.41,E2 -5347.41} C_VEL
LIN {X 0,Y 510.343,Z 158.112,A -85,B 0,C 180,E1 -5347.62,E2 -5347.62} C_VEL
LIN {X 0,Y 510.583,Z 141.453,A -85,B 0,C 180,E1 -5350.796,E2 -5350.796} C_VEL
LIN {X 0,Y 510.004,Z 135.724,A -85,B 0,C 180,E1 -5351.916,E2 -5351.916} C_VEL
LIN {X 0,Y 509.906,Z 134.973,A -85,B 0,C 180,E1 -5352.081,E2 -5352.081} C_VEL
LIN {X 0,Y 509.853,Z 134.975,A -85,B 0,C 180,E1 -5355.333,E2 -5355.333} C_VEL
LIN {X 0,Y 509.863,Z 134.973,A -85,B 0,C 180,E1 -5358.576,E2 -5358.576} C_VEL
LIN {X 0,Y 509.85,Z 134.982,A -85,B 0,C 180,E1 -5361.787,E2 -5361.787} C_VEL
LIN {X 0,Y 509.827,Z 134.975,A -85,B 0,C 180,E1 -5364.623,E2 -5364.623} C_VEL
LIN {X 0,Y 509.859,Z 134.979,A -85,B 0,C 180,E1 -5367.482,E2 -5367.482} C_VEL
LIN {X 0,Y 509.857,Z 134.97,A -85,B 0,C 180,E1 -5370.274,E2 -5370.274} C_VEL
LIN {X 0,Y 509.883,Z 134.971,A -85,B 0,C 180,E1 -5372.945,E2 -5372.945} C_VEL
LIN {X 0,Y 509.864,Z 134.974,A -85,B 0,C 180,E1 -5375.575,E2 -5375.575} C_VEL
LIN {X 0,Y 509.85,Z 134.978,A -85,B 0,C 180,E1 -5378.999,E2 -5378.999} C_VEL
LIN {X 0,Y 509.857,Z 134.973,A -85,B 0,C 180,E1 -5381.517,E2 -5381.517} C_VEL
LIN {X 0,Y 509.912,Z 134.971,A -85,B 0,C 180,E1 -5384.82,E2 -5384.82} C_VEL
LIN {X 0,Y 509.902,Z 134.965,A -85,B 0,C 180,E1 -5388.125,E2 -5388.125} C_VEL
LIN {X 0,Y 509.905,Z 134.964,A -85,B 0,C 180,E1 -5391.28,E2 -5391.28} C_VEL
LIN {X 0,Y 509.976,Z 134.962,A -85,B 0,C 180,E1 -5394.465,E2 -5394.465} C_VEL
LIN {X 0,Y 510.052,Z 134.945,A -85,B 0,C 180,E1 -5397.632,E2 -5397.632} C_VEL
LIN {X 0,Y 510.041,Z 134.947,A -85,B 0,C 180,E1 -5400.79,E2 -5400.79} C_VEL
LIN {X 0,Y 510.047,Z 134.952,A -85,B 0,C 180,E1 -5402.37,E2 -5402.37} C_VEL
LIN {X 0,Y 509.964,Z 134.954,A -85,B 0,C 180,E1 -5405.537,E2 -5405.537} C_VEL
LIN {X 0,Y 509.891,Z 134.967,A -85,B 0,C 180,E1 -5408.721,E2 -5408.721} C_VEL
LIN {X 0,Y 509.907,Z 134.966,A -85,B 0,C 180,E1 -5411.932,E2 -5411.932} C_VEL
LIN {X 0,Y 509.898,Z 134.965,A -85,B 0,C 180,E1 -5415.242,E2 -5415.242} C_VEL
LIN {X 0,Y 509.835,Z 134.974,A -85,B 0,C 180,E1 -5418.485,E2 -5418.485} C_VEL
LIN {X 0,Y 509.825,Z 134.973,A -85,B 0,C 180,E1 -5421.003,E2 -5421.003} C_VEL
LIN {X 0,Y 509.81,Z 134.983,A -85,B 0,C 180,E1 -5423.565,E2 -5423.565} C_VEL
LIN {X 0,Y 509.817,Z 134.973,A -85,B 0,C 180,E1 -5426.356,E2 -5426.356} C_VEL
LIN {X 0,Y 509.795,Z 134.98,A -85,B 0,C 180,E1 -5428.85,E2 -5428.85} C_VEL
LIN {X 0,Y 509.79,Z 134.985,A -85,B 0,C 180,E1 -5431.593,E2 -5431.593} C_VEL
LIN {X 0,Y 509.822,Z 134.973,A -85,B 0,C 180,E1 -5434.416,E2 -5434.416} C_VEL
LIN {X 0,Y 509.765,Z 134.987,A -85,B 0,C 180,E1 -5437.346,E2 -5437.346} C_VEL
LIN {X 0,Y 509.788,Z 134.981,A -85,B 0,C 180,E1 -5440.388,E2 -5440.388} C_VEL
LIN {X 0,Y 509.794,Z 134.98,A -85,B 0,C 180,E1 -5443.575,E2 -5443.575} C_VEL
LIN {X 0,Y 509.794,Z 134.984,A -85,B 0,C 180,E1 -5446.425,E2 -5446.425} C_VEL
LIN {X 0,Y 509.814,Z 134.978,A -85,B 0,C 180,E1 -5449.615,E2 -5449.615} C_VEL
LIN {X 0,Y 509.808,Z 134.983,A -85,B 0,C 180,E1 -5452.658,E2 -5452.658} C_VEL
LIN {X 0,Y 509.841,Z 134.974,A -85,B 0,C 180,E1 -5455.801,E2 -5455.801} C_VEL
LIN {X 0,Y 509.846,Z 134.979,A -85,B 0,C 180,E1 -5458.721,E2 -5458.721} C_VEL
LIN {X 0,Y 509.839,Z 134.975,A -85,B 0,C 180,E1 -5461.153,E2 -5461.153} C_VEL
LIN {X 0,Y 509.852,Z 134.977,A -85,B 0,C 180,E1 -5463.826,E2 -5463.826} C_VEL
LIN {X 0,Y 509.868,Z 135.16,A -85,B 0,C 180,E1 -5465.219,E2 -5465.219} C_VEL
LIN {X 0,Y 511.281,Z 142.669,A -85,B 0,C 180,E1 -5466.507,E2 -5466.507} C_VEL
LIN {X 0,Y 511.312,Z 149.276,A -85,B 0,C 180,E1 -5467.578,E2 -5467.578} C_VEL
LIN {X 0,Y 510.859,Z 165.096,A -85,B 0,C 180,E1 -5470.093,E2 -5470.093} C_VEL
LIN {X 0,Y 510.465,Z 180.883,A -85,B 0,C 180,E1 -5472.575,E2 -5472.575} C_VEL
LIN {X 0,Y 510.221,Z 192.648,A -85,B 0,C 180,E1 -5474.41,E2 -5474.41} C_VEL
LIN {X 0,Y 512.149,Z 206.107,A -85,B 0,C 180,E1 -5474.666,E2 -5474.666} C_VEL
LIN {X 0,Y 511.721,Z 300.663,A -85,B 0,C 180,E1 -5476.017,E2 -5476.017} C_VEL
LIN {X 0,Y 511.494,Z 313.337,A -85,B 0,C 180,E1 -5476.34,E2 -5476.34} C_VEL
LIN {X 0,Y 511.167,Z 326.35,A -85,B 0,C 180,E1 -5476.837,E2 -5476.837} C_VEL
LIN {X 0,Y 510.83,Z 337.992,A -85,B 0,C 180,E1 -5477.442,E2 -5477.442} C_VEL
LIN {X 0,Y 510.511,Z 349.058,A -85,B 0,C 180,E1 -5478.184,E2 -5478.184} C_VEL
LIN {X 0,Y 510.231,Z 359.77,A -85,B 0,C 180,E1 -5479.083,E2 -5479.083} C_VEL
LIN {X 0,Y 509.853,Z 369.418,A -85,B 0,C 180,E1 -5480.078,E2 -5480.078} C_VEL
LIN {X 0,Y 509.649,Z 377.333,A -85,B 0,C 180,E1 -5481.075,E2 -5481.075} C_VEL
LIN {X 0,Y 509.452,Z 385.063,A -85,B 0,C 180,E1 -5482.27,E2 -5482.27} C_VEL
LIN {X 0,Y 509.289,Z 392.188,A -85,B 0,C 180,E1 -5483.662,E2 -5483.662} C_VEL
LIN {X 0,Y 509.241,Z 396.931,A -85,B 0,C 180,E1 -5484.853,E2 -5484.853} C_VEL
LIN {X 0,Y 509.245,Z 400.556,A -85,B 0,C 180,E1 -5486.043,E2 -5486.043} C_VEL
LIN {X 0,Y 509.201,Z 402.425,A -85,B 0,C 180,E1 -5486.835,E2 -5486.835} C_VEL
LIN {X 0,Y 509.19,Z 403.827,A -85,B 0,C 180,E1 -5487.627,E2 -5487.627} C_VEL
LIN {X 0,Y 509.079,Z 405.437,A -85,B 0,C 180,E1 -5489.209,E2 -5489.209} C_VEL
LIN {X 0,Y 509.075,Z 405.656,A -85,B 0,C 180,E1 -5490,E2 -5490} C_VEL
LIN {X 0,Y 509.113,Z 404.836,A -85,B 0,C 180,E1 -5491.582,E2 -5491.582} C_VEL
LIN {X 0,Y 509.19,Z 403.843,A -85,B 0,C 180,E1 -5492.373,E2 -5492.373} C_VEL
LIN {X 0,Y 509.201,Z 402.446,A -85,B 0,C 180,E1 -5493.165,E2 -5493.165} C_VEL
LIN {X 0,Y 509.202,Z 399.504,A -85,B 0,C 180,E1 -5494.354,E2 -5494.354} C_VEL
LIN {X 0,Y 509.283,Z 395.524,A -85,B 0,C 180,E1 -5495.544,E2 -5495.544} C_VEL
LIN {X 0,Y 509.367,Z 389.498,A -85,B 0,C 180,E1 -5496.914,E2 -5496.914} C_VEL
LIN {X 0,Y 509.495,Z 382.702,A -85,B 0,C 180,E1 -5498.128,E2 -5498.128} C_VEL
LIN {X 0,Y 509.733,Z 374.399,A -85,B 0,C 180,E1 -5499.323,E2 -5499.323} C_VEL
LIN {X 0,Y 509.969,Z 365.883,A -85,B 0,C 180,E1 -5500.321,E2 -5500.321} C_VEL
LIN {X 0,Y 510.334,Z 355.365,A -85,B 0,C 180,E1 -5501.318,E2 -5501.318} C_VEL
LIN {X 0,Y 510.647,Z 344.314,A -85,B 0,C 180,E1 -5502.161,E2 -5502.161} C_VEL
LIN {X 0,Y 510.986,Z 333.545,A -85,B 0,C 180,E1 -5502.814,E2 -5502.814} C_VEL
LIN {X 0,Y 511.258,Z 321.802,A -85,B 0,C 180,E1 -5503.363,E2 -5503.363} C_VEL
LIN {X 0,Y 511.582,Z 308.273,A -85,B 0,C 180,E1 -5503.81,E2 -5503.81} C_VEL
LIN {X 0,Y 511.793,Z 294.735,A -85,B 0,C 180,E1 -5504.083,E2 -5504.083} C_VEL
LIN {X 0,Y 512.097,Z 205.177,A -85,B 0,C 180,E1 -5505.351,E2 -5505.351} C_VEL
LIN {X 0,Y 510.239,Z 192.742,A -85,B 0,C 180,E1 -5505.603,E2 -5505.603} C_VEL
LIN {X 0,Y 510.726,Z 173.283,A -85,B 0,C 180,E1 -5508.659,E2 -5508.659} C_VEL
LIN {X 0,Y 511.221,Z 154.959,A -85,B 0,C 180,E1 -5511.577,E2 -5511.577} C_VEL
LIN {X 0,Y 511.417,Z 143.154,A -85,B 0,C 180,E1 -5513.486,E2 -5513.486} C_VEL
LIN {X 0,Y 509.845,Z 134.978,A -85,B 0,C 180,E1 -5514.921,E2 -5514.921} C_VEL
LIN {X 0,Y 509.837,Z 134.979,A -85,B 0,C 180,E1 -5517.949,E2 -5517.949} C_VEL
LIN {X 0,Y 509.838,Z 134.975,A -85,B 0,C 180,E1 -5520.667,E2 -5520.667} C_VEL
LIN {X 0,Y 509.843,Z 134.979,A -85,B 0,C 180,E1 -5523.463,E2 -5523.463} C_VEL
LIN {X 0,Y 509.813,Z 134.976,A -85,B 0,C 180,E1 -5526.355,E2 -5526.355} C_VEL
LIN {X 0,Y 509.837,Z 134.98,A -85,B 0,C 180,E1 -5529.354,E2 -5529.354} C_VEL
LIN {X 0,Y 509.795,Z 134.978,A -85,B 0,C 180,E1 -5532.494,E2 -5532.494} C_VEL
LIN {X 0,Y 509.844,Z 134.98,A -85,B 0,C 180,E1 -5535.33,E2 -5535.33} C_VEL
LIN {X 0,Y 509.812,Z 134.977,A -85,B 0,C 180,E1 -5538.57,E2 -5538.57} C_VEL
LIN {X 0,Y 509.854,Z 134.972,A -85,B 0,C 180,E1 -5541.787,E2 -5541.787} C_VEL
LIN {X 0,Y 509.829,Z 134.976,A -85,B 0,C 180,E1 -5544.621,E2 -5544.621} C_VEL
LIN {X 0,Y 509.863,Z 134.972,A -85,B 0,C 180,E1 -5547.48,E2 -5547.48} C_VEL
LIN {X 0,Y 509.833,Z 134.974,A -85,B 0,C 180,E1 -5550.28,E2 -5550.28} C_VEL
LIN {X 0,Y 509.83,Z 134.981,A -85,B 0,C 180,E1 -5552.941,E2 -5552.941} C_VEL
LIN {X 0,Y 509.839,Z 134.973,A -85,B 0,C 180,E1 -5555.572,E2 -5555.572} C_VEL
LIN {X 0,Y 509.815,Z 134.977,A -85,B 0,C 180,E1 -5558.148,E2 -5558.148} C_VEL
LIN {X 0,Y 509.85,Z 134.98,A -85,B 0,C 180,E1 -5560.68,E2 -5560.68} C_VEL
LIN {X 0,Y 509.79,Z 134.98,A -85,B 0,C 180,E1 -5563.171,E2 -5563.171} C_VEL
LIN {X 0,Y 509.846,Z 134.971,A -85,B 0,C 180,E1 -5565.633,E2 -5565.633} C_VEL
LIN {X 0,Y 509.916,Z 134.966,A -85,B 0,C 180,E1 -5568.874,E2 -5568.874} C_VEL
LIN {X 0,Y 509.883,Z 134.971,A -85,B 0,C 180,E1 -5572.077,E2 -5572.077} C_VEL
LIN {X 0,Y 509.941,Z 134.967,A -85,B 0,C 180,E1 -5574.463,E2 -5574.463} C_VEL
LIN {X 0,Y 510.045,Z 134.948,A -85,B 0,C 180,E1 -5577.63,E2 -5577.63} C_VEL
LIN {X 0,Y 510.038,Z 134.953,A -85,B 0,C 180,E1 -5579.999,E2 -5579.999} C_VEL
LIN {X 0,Y 510.045,Z 134.952,A -85,B 0,C 180,E1 -5582.368,E2 -5582.368} C_VEL
LIN {X 0,Y 509.939,Z 134.962,A -85,B 0,C 180,E1 -5585.535,E2 -5585.535} C_VEL
LIN {X 0,Y 509.878,Z 134.975,A -85,B 0,C 180,E1 -5587.922,E2 -5587.922} C_VEL
LIN {X 0,Y 509.865,Z 134.969,A -85,B 0,C 180,E1 -5591.126,E2 -5591.126} C_VEL
LIN {X 0,Y 509.829,Z 134.977,A -85,B 0,C 180,E1 -5593.552,E2 -5593.552} C_VEL
LIN {X 0,Y 509.798,Z 134.984,A -85,B 0,C 180,E1 -5596.004,E2 -5596.004} C_VEL
LIN {X 0,Y 509.829,Z 134.974,A -85,B 0,C 180,E1 -5598.484,E2 -5598.484} C_VEL
LIN {X 0,Y 509.819,Z 134.975,A -85,B 0,C 180,E1 -5601.002,E2 -5601.002} C_VEL
LIN {X 0,Y 509.81,Z 134.983,A -85,B 0,C 180,E1 -5603.564,E2 -5603.564} C_VEL
LIN {X 0,Y 509.815,Z 134.976,A -85,B 0,C 180,E1 -5606.355,E2 -5606.355} C_VEL
LIN {X 0,Y 509.823,Z 134.975,A -85,B 0,C 180,E1 -5608.847,E2 -5608.847} C_VEL
LIN {X 0,Y 509.81,Z 134.983,A -85,B 0,C 180,E1 -5611.59,E2 -5611.59} C_VEL
LIN {X 0,Y 509.832,Z 134.973,A -85,B 0,C 180,E1 -5614.414,E2 -5614.414} C_VEL
LIN {X 0,Y 509.803,Z 134.986,A -85,B 0,C 180,E1 -5617.341,E2 -5617.341} C_VEL
LIN {X 0,Y 509.809,Z 134.976,A -85,B 0,C 180,E1 -5620.384,E2 -5620.384} C_VEL
LIN {X 0,Y 509.802,Z 134.98,A -85,B 0,C 180,E1 -5623.573,E2 -5623.573} C_VEL
LIN {X 0,Y 509.801,Z 134.978,A -85,B 0,C 180,E1 -5626.426,E2 -5626.426} C_VEL
LIN {X 0,Y 509.808,Z 134.978,A -85,B 0,C 180,E1 -5629.614,E2 -5629.614} C_VEL
LIN {X 0,Y 509.801,Z 134.981,A -85,B 0,C 180,E1 -5632.657,E2 -5632.657} C_VEL
LIN {X 0,Y 509.795,Z 134.978,A -85,B 0,C 180,E1 -5633.697,E2 -5633.697} C_VEL
LIN {X 0,Y 509.128,Z 135.063,A -85,B 0,C 180,E1 -5634.357,E2 -5634.357} C_VEL
LIN {X 0,Y 506.308,Z 135.419,A -85,B 0,C 180,E1 -5635.429,E2 -5635.429} C_VEL
LIN {X 0,Y 503.918,Z 135.719,A -85,B 0,C 180,E1 -5636.292,E2 -5636.292} C_VEL
LIN {X 0,Y 502.876,Z 135.847,A -85,B 0,C 180,E1 -5636.959,E2 -5636.959} C_VEL
LIN {X 0,Y 502.782,Z 135.855,A -85,B 0,C 180,E1 -5637.184,E2 -5637.184} C_VEL
LIN {X 0,Y 502.785,Z 135.852,A -85,B 0,C 180,E1 -5640.069,E2 -5640.069} C_VEL
LIN {X 0,Y 502.777,Z 135.853,A -85,B 0,C 180,E1 -5643.429,E2 -5643.429} C_VEL
LIN {X 0,Y 502.753,Z 135.857,A -85,B 0,C 180,E1 -5646.084,E2 -5646.084} C_VEL
LIN {X 0,Y 502.823,Z 135.846,A -85,B 0,C 180,E1 -5649.463,E2 -5649.463} C_VEL
LIN {X 0,Y 502.777,Z 135.855,A -85,B 0,C 180,E1 -5652.09,E2 -5652.09} C_VEL
LIN {X 0,Y 502.818,Z 135.847,A -85,B 0,C 180,E1 -5655.428,E2 -5655.428} C_VEL
LIN {X 0,Y 502.829,Z 135.849,A -85,B 0,C 180,E1 -5658.715,E2 -5658.715} C_VEL
LIN {X 0,Y 502.838,Z 135.849,A -85,B 0,C 180,E1 -5661.965,E2 -5661.965} C_VEL
LIN {X 0,Y 502.884,Z 135.845,A -85,B 0,C 180,E1 -5664.386,E2 -5664.386} C_VEL
LIN {X 0,Y 503.001,Z 135.828,A -85,B 0,C 180,E1 -5667.597,E2 -5667.597} C_VEL
LIN {X 0,Y 502.995,Z 135.834,A -85,B 0,C 180,E1 -5670,E2 -5670} C_VEL
LIN {X 0,Y 502.942,Z 136.014,A -85,B 0,C 180,E1 -5671.852,E2 -5671.852} C_VEL
LIN {X 0,Y 503.51,Z 142.687,A -85,B 0,C 180,E1 -5673.2,E2 -5673.2} C_VEL
LIN {X 0,Y 503.319,Z 158.463,A -85,B 0,C 180,E1 -5676.263,E2 -5676.263} C_VEL
LIN {X 0,Y 505.468,Z 170.745,A -85,B 0,C 180,E1 -5676.511,E2 -5676.511} C_VEL
LIN {X 0,Y 504.868,Z 264.905,A -85,B 0,C 180,E1 -5677.876,E2 -5677.876} C_VEL
LIN {X 0,Y 504.612,Z 278.2,A -85,B 0,C 180,E1 -5678.228,E2 -5678.228} C_VEL
LIN {X 0,Y 504.384,Z 291.248,A -85,B 0,C 180,E1 -5678.75,E2 -5678.75} C_VEL
LIN {X 0,Y 504.087,Z 303.554,A -85,B 0,C 180,E1 -5679.429,E2 -5679.429} C_VEL
LIN {X 0,Y 503.708,Z 315.06,A -85,B 0,C 180,E1 -5680.247,E2 -5680.247} C_VEL
LIN {X 0,Y 503.402,Z 325.397,A -85,B 0,C 180,E1 -5681.169,E2 -5681.169} C_VEL
LIN {X 0,Y 503.072,Z 333.883,A -85,B 0,C 180,E1 -5682.096,E2 -5682.096} C_VEL
LIN {X 0,Y 502.736,Z 343.079,A -85,B 0,C 180,E1 -5683.336,E2 -5683.336} C_VEL
LIN {X 0,Y 502.495,Z 350.491,A -85,B 0,C 180,E1 -5684.581,E2 -5684.581} C_VEL
LIN {X 0,Y 502.342,Z 356.39,A -85,B 0,C 180,E1 -5685.832,E2 -5685.832} C_VEL
LIN {X 0,Y 502.211,Z 361.015,A -85,B 0,C 180,E1 -5687.09,E2 -5687.09} C_VEL
LIN {X 0,Y 502.14,Z 363.454,A -85,B 0,C 180,E1 -5687.934,E2 -5687.934} C_VEL
LIN {X 0,Y 502.089,Z 365.442,A -85,B 0,C 180,E1 -5688.78,E2 -5688.78} C_VEL
LIN {X 0,Y 502.034,Z 367.776,A -85,B 0,C 180,E1 -5690.295,E2 -5690.295} C_VEL
LIN {X 0,Y 501.997,Z 368.585,A -85,B 0,C 180,E1 -5691.346,E2 -5691.346} C_VEL
LIN {X 0,Y 502.007,Z 368.66,A -85,B 0,C 180,E1 -5692.486,E2 -5692.486} C_VEL
LIN {X 0,Y 502.022,Z 367.63,A -85,B 0,C 180,E1 -5693.953,E2 -5693.953} C_VEL
LIN {X 0,Y 502.037,Z 366.339,A -85,B 0,C 180,E1 -5694.833,E2 -5694.833} C_VEL
LIN {X 0,Y 502.124,Z 364.568,A -85,B 0,C 180,E1 -5695.715,E2 -5695.715} C_VEL
LIN {X 0,Y 502.24,Z 360.894,A -85,B 0,C 180,E1 -5697.051,E2 -5697.051} C_VEL
LIN {X 0,Y 502.338,Z 355.816,A -85,B 0,C 180,E1 -5698.404,E2 -5698.404} C_VEL
LIN {X 0,Y 502.508,Z 350.058,A -85,B 0,C 180,E1 -5699.598,E2 -5699.598} C_VEL
LIN {X 0,Y 502.763,Z 342.096,A -85,B 0,C 180,E1 -5700.912,E2 -5700.912} C_VEL
LIN {X 0,Y 503.09,Z 333.387,A -85,B 0,C 180,E1 -5702.063,E2 -5702.063} C_VEL
LIN {X 0,Y 503.435,Z 323.48,A -85,B 0,C 180,E1 -5703.114,E2 -5703.114} C_VEL
LIN {X 0,Y 503.799,Z 312.721,A -85,B 0,C 180,E1 -5704.035,E2 -5704.035} C_VEL
LIN {X 0,Y 504.173,Z 301.721,A -85,B 0,C 180,E1 -5704.783,E2 -5704.783} C_VEL
LIN {X 0,Y 504.53,Z 289.13,A -85,B 0,C 180,E1 -5705.438,E2 -5705.438} C_VEL
LIN {X 0,Y 504.745,Z 276.374,A -85,B 0,C 180,E1 -5705.925,E2 -5705.925} C_VEL
LIN {X 0,Y 504.899,Z 264.096,A -85,B 0,C 180,E1 -5706.232,E2 -5706.232} C_VEL
LIN {X 0,Y 505.384,Z 168.998,A -85,B 0,C 180,E1 -5707.612,E2 -5707.612} C_VEL
LIN {X 0,Y 503.372,Z 158.297,A -85,B 0,C 180,E1 -5707.854,E2 -5707.854} C_VEL
LIN {X 0,Y 503.622,Z 143.374,A -85,B 0,C 180,E1 -5710.722,E2 -5710.722} C_VEL
LIN {X 0,Y 503.358,Z 138.535,A -85,B 0,C 180,E1 -5711.667,E2 -5711.667} C_VEL
LIN {X 0,Y 502.878,Z 135.848,A -85,B 0,C 180,E1 -5712.242,E2 -5712.242} C_VEL
LIN {X 0,Y 502.786,Z 135.857,A -85,B 0,C 180,E1 -5715.662,E2 -5715.662} C_VEL
LIN {X 0,Y 502.832,Z 135.854,A -85,B 0,C 180,E1 -5717.866,E2 -5717.866} C_VEL
LIN {X 0,Y 502.807,Z 135.851,A -85,B 0,C 180,E1 -5721.026,E2 -5721.026} C_VEL
LIN {X 0,Y 502.772,Z 135.857,A -85,B 0,C 180,E1 -5724.17,E2 -5724.17} C_VEL
LIN {X 0,Y 502.83,Z 135.848,A -85,B 0,C 180,E1 -5726.994,E2 -5726.994} C_VEL
LIN {X 0,Y 502.813,Z 135.849,A -85,B 0,C 180,E1 -5730.066,E2 -5730.066} C_VEL
LIN {X 0,Y 502.831,Z 135.847,A -85,B 0,C 180,E1 -5732.534,E2 -5732.534} C_VEL
LIN {X 0,Y 502.826,Z 135.854,A -85,B 0,C 180,E1 -5735.3,E2 -5735.3} C_VEL
LIN {X 0,Y 502.78,Z 135.854,A -85,B 0,C 180,E1 -5737.827,E2 -5737.827} C_VEL
LIN {X 0,Y 502.82,Z 135.849,A -85,B 0,C 180,E1 -5740.401,E2 -5740.401} C_VEL
LIN {X 0,Y 502.811,Z 135.854,A -85,B 0,C 180,E1 -5742.932,E2 -5742.932} C_VEL
LIN {X 0,Y 502.842,Z 135.846,A -85,B 0,C 180,E1 -5745.43,E2 -5745.43} C_VEL
LIN {X 0,Y 502.878,Z 135.847,A -85,B 0,C 180,E1 -5748.718,E2 -5748.718} C_VEL
LIN {X 0,Y 502.882,Z 135.837,A -85,B 0,C 180,E1 -5751.967,E2 -5751.967} C_VEL
LIN {X 0,Y 502.93,Z 135.838,A -85,B 0,C 180,E1 -5754.387,E2 -5754.387} C_VEL
LIN {X 0,Y 503.021,Z 135.821,A -85,B 0,C 180,E1 -5757.598,E2 -5757.598} C_VEL
LIN {X 0,Y 502.992,Z 135.825,A -85,B 0,C 180,E1 -5760.801,E2 -5760.801} C_VEL
LIN {X 0,Y 503.014,Z 135.829,A -85,B 0,C 180,E1 -5762.403,E2 -5762.403} C_VEL
LIN {X 0,Y 502.917,Z 135.832,A -85,B 0,C 180,E1 -5765.614,E2 -5765.614} C_VEL
LIN {X 0,Y 502.854,Z 135.843,A -85,B 0,C 180,E1 -5768.844,E2 -5768.844} C_VEL
LIN {X 0,Y 502.848,Z 135.849,A -85,B 0,C 180,E1 -5772.102,E2 -5772.102} C_VEL
LIN {X 0,Y 502.849,Z 135.845,A -85,B 0,C 180,E1 -5775.4,E2 -5775.4} C_VEL
LIN {X 0,Y 502.808,Z 135.849,A -85,B 0,C 180,E1 -5778.753,E2 -5778.753} C_VEL
LIN {X 0,Y 502.764,Z 135.855,A -85,B 0,C 180,E1 -5781.313,E2 -5781.313} C_VEL
LIN {X 0,Y 502.763,Z 135.859,A -85,B 0,C 180,E1 -5783.916,E2 -5783.916} C_VEL
LIN {X 0,Y 502.785,Z 135.849,A -85,B 0,C 180,E1 -5786.571,E2 -5786.571} C_VEL
LIN {X 0,Y 502.754,Z 135.862,A -85,B 0,C 180,E1 -5789.293,E2 -5789.293} C_VEL
LIN {X 0,Y 502.758,Z 135.856,A -85,B 0,C 180,E1 -5792.087,E2 -5792.087} C_VEL
LIN {X 0,Y 502.754,Z 135.858,A -85,B 0,C 180,E1 -5794.97,E2 -5794.97} C_VEL
LIN {X 0,Y 502.75,Z 135.856,A -85,B 0,C 180,E1 -5798.479,E2 -5798.479} C_VEL
LIN {X 0,Y 502.752,Z 135.863,A -85,B 0,C 180,E1 -5801.073,E2 -5801.073} C_VEL
LIN {X 0,Y 502.78,Z 135.856,A -85,B 0,C 180,E1 -5804.529,E2 -5804.529} C_VEL
LIN {X 0,Y 502.768,Z 135.856,A -85,B 0,C 180,E1 -5807.858,E2 -5807.858} C_VEL
LIN {X 0,Y 502.786,Z 135.857,A -85,B 0,C 180,E1 -5811.022,E2 -5811.022} C_VEL
LIN {X 0,Y 502.768,Z 135.855,A -85,B 0,C 180,E1 -5814.171,E2 -5814.171} C_VEL
LIN {X 0,Y 502.806,Z 135.853,A -85,B 0,C 180,E1 -5816.999,E2 -5816.999} C_VEL
LIN {X 0,Y 502.813,Z 135.854,A -85,B 0,C 180,E1 -5820.066,E2 -5820.066} C_VEL
LIN {X 0,Y 502.777,Z 135.857,A -85,B 0,C 180,E1 -5823.46,E2 -5823.46} C_VEL
LIN {X 0,Y 502.822,Z 136.059,A -85,B 0,C 180,E1 -5825.043,E2 -5825.043} C_VEL
LIN {X 0,Y 504.43,Z 144.813,A -85,B 0,C 180,E1 -5826.565,E2 -5826.565} C_VEL
LIN {X 0,Y 504.107,Z 158.241,A -85,B 0,C 180,E1 -5828.748,E2 -5828.748} C_VEL
LIN {X 0,Y 503.588,Z 176.962,A -85,B 0,C 180,E1 -5831.746,E2 -5831.746} C_VEL
LIN {X 0,Y 503.203,Z 192.339,A -85,B 0,C 180,E1 -5834.181,E2 -5834.181} C_VEL
LIN {X 0,Y 505.319,Z 207.262,A -85,B 0,C 180,E1 -5834.473,E2 -5834.473} C_VEL
LIN {X 0,Y 504.798,Z 301.522,A -85,B 0,C 180,E1 -5835.847,E2 -5835.847} C_VEL
LIN {X 0,Y 504.517,Z 315.333,A -85,B 0,C 180,E1 -5836.225,E2 -5836.225} C_VEL
LIN {X 0,Y 504.213,Z 327.194,A -85,B 0,C 180,E1 -5836.704,E2 -5836.704} C_VEL
LIN {X 0,Y 503.855,Z 338.284,A -85,B 0,C 180,E1 -5837.3,E2 -5837.3} C_VEL
LIN {X 0,Y 503.512,Z 350.076,A -85,B 0,C 180,E1 -5838.119,E2 -5838.119} C_VEL
LIN {X 0,Y 503.199,Z 360.568,A -85,B 0,C 180,E1 -5839.03,E2 -5839.03} C_VEL
LIN {X 0,Y 502.823,Z 369.142,A -85,B 0,C 180,E1 -5839.938,E2 -5839.938} C_VEL
LIN {X 0,Y 502.605,Z 377.06,A -85,B 0,C 180,E1 -5840.949,E2 -5840.949} C_VEL
LIN {X 0,Y 502.375,Z 384.793,A -85,B 0,C 180,E1 -5842.161,E2 -5842.161} C_VEL
LIN {X 0,Y 502.237,Z 391.511,A -85,B 0,C 180,E1 -5843.482,E2 -5843.482} C_VEL
LIN {X 0,Y 502.171,Z 396.666,A -85,B 0,C 180,E1 -5844.781,E2 -5844.781} C_VEL
LIN {X 0,Y 502.138,Z 400.292,A -85,B 0,C 180,E1 -5845.987,E2 -5845.987} C_VEL
LIN {X 0,Y 502.12,Z 402.163,A -85,B 0,C 180,E1 -5846.791,E2 -5846.791} C_VEL
LIN {X 0,Y 502.092,Z 403.566,A -85,B 0,C 180,E1 -5847.593,E2 -5847.593} C_VEL
LIN {X 0,Y 501.996,Z 405.178,A -85,B 0,C 180,E1 -5849.198,E2 -5849.198} C_VEL
LIN {X 0,Y 501.989,Z 405.398,A -85,B 0,C 180,E1 -5850,E2 -5850} C_VEL
LIN {X 0,Y 502.037,Z 404.579,A -85,B 0,C 180,E1 -5851.605,E2 -5851.605} C_VEL
LIN {X 0,Y 502.092,Z 403.585,A -85,B 0,C 180,E1 -5852.407,E2 -5852.407} C_VEL
LIN {X 0,Y 502.121,Z 402.187,A -85,B 0,C 180,E1 -5853.21,E2 -5853.21} C_VEL
LIN {X 0,Y 502.1,Z 399.245,A -85,B 0,C 180,E1 -5854.415,E2 -5854.415} C_VEL
LIN {X 0,Y 502.198,Z 395.264,A -85,B 0,C 180,E1 -5855.622,E2 -5855.622} C_VEL
LIN {X 0,Y 502.292,Z 389.237,A -85,B 0,C 180,E1 -5857.012,E2 -5857.012} C_VEL
LIN {X 0,Y 502.448,Z 382.44,A -85,B 0,C 180,E1 -5858.243,E2 -5858.243} C_VEL
LIN {X 0,Y 502.706,Z 374.135,A -85,B 0,C 180,E1 -5859.455,E2 -5859.455} C_VEL
LIN {X 0,Y 502.958,Z 365.617,A -85,B 0,C 180,E1 -5860.466,E2 -5860.466} C_VEL
LIN {X 0,Y 503.348,Z 355.094,A -85,B 0,C 180,E1 -5861.477,E2 -5861.477} C_VEL
LIN {X 0,Y 503.661,Z 344.038,A -85,B 0,C 180,E1 -5862.332,E2 -5862.332} C_VEL
LIN {X 0,Y 504.034,Z 333.263,A -85,B 0,C 180,E1 -5862.994,E2 -5862.994} C_VEL
LIN {X 0,Y 504.353,Z 321.507,A -85,B 0,C 180,E1 -5863.549,E2 -5863.549} C_VEL
LIN {X 0,Y 504.704,Z 307.962,A -85,B 0,C 180,E1 -5864.002,E2 -5864.002} C_VEL
LIN {X 0,Y 504.92,Z 294.37,A -85,B 0,C 180,E1 -5864.278,E2 -5864.278} C_VEL
LIN {X 0,Y 505.212,Z 205.886,A -85,B 0,C 180,E1 -5865.551,E2 -5865.551} C_VEL
LIN {X 0,Y 503.218,Z 192.544,A -85,B 0,C 180,E1 -5865.817,E2 -5865.817} C_VEL
LIN {X 0,Y 503.738,Z 174.34,A -85,B 0,C 180,E1 -5868.717,E2 -5868.717} C_VEL
LIN {X 0,Y 504.27,Z 156.015,A -85,B 0,C 180,E1 -5871.675,E2 -5871.675} C_VEL
LIN {X 0,Y 504.523,Z 145.248,A -85,B 0,C 180,E1 -5873.438,E2 -5873.438} C_VEL
LIN {X 0,Y 502.788,Z 135.857,A -85,B 0,C 180,E1 -5875.113,E2 -5875.113} C_VEL
LIN {X 0,Y 502.776,Z 135.855,A -85,B 0,C 180,E1 -5878.28,E2 -5878.28} C_VEL
LIN {X 0,Y 502.796,Z 135.855,A -85,B 0,C 180,E1 -5881.144,E2 -5881.144} C_VEL
LIN {X 0,Y 502.79,Z 135.853,A -85,B 0,C 180,E1 -5883.995,E2 -5883.995} C_VEL
LIN {X 0,Y 502.768,Z 135.857,A -85,B 0,C 180,E1 -5887.176,E2 -5887.176} C_VEL
LIN {X 0,Y 502.775,Z 135.854,A -85,B 0,C 180,E1 -5890.017,E2 -5890.017} C_VEL
LIN {X 0,Y 502.752,Z 135.862,A -85,B 0,C 180,E1 -5893.234,E2 -5893.234} C_VEL
LIN {X 0,Y 502.783,Z 135.855,A -85,B 0,C 180,E1 -5895.66,E2 -5895.66} C_VEL
LIN {X 0,Y 502.77,Z 135.859,A -85,B 0,C 180,E1 -5899.012,E2 -5899.012} C_VEL
LIN {X 0,Y 502.794,Z 135.85,A -85,B 0,C 180,E1 -5902.046,E2 -5902.046} C_VEL
LIN {X 0,Y 502.796,Z 135.858,A -85,B 0,C 180,E1 -5905.033,E2 -5905.033} C_VEL
LIN {X 0,Y 502.783,Z 135.851,A -85,B 0,C 180,E1 -5907.915,E2 -5907.915} C_VEL
LIN {X 0,Y 502.795,Z 135.855,A -85,B 0,C 180,E1 -5910.71,E2 -5910.71} C_VEL
LIN {X 0,Y 502.78,Z 135.853,A -85,B 0,C 180,E1 -5913.459,E2 -5913.459} C_VEL
LIN {X 0,Y 502.766,Z 135.854,A -85,B 0,C 180,E1 -5916.084,E2 -5916.084} C_VEL
LIN {X 0,Y 502.836,Z 135.845,A -85,B 0,C 180,E1 -5919.464,E2 -5919.464} C_VEL
LIN {X 0,Y 502.79,Z 135.852,A -85,B 0,C 180,E1 -5922.09,E2 -5922.09} C_VEL
LIN {X 0,Y 502.828,Z 135.846,A -85,B 0,C 180,E1 -5925.428,E2 -5925.428} C_VEL
LIN {X 0,Y 502.881,Z 135.845,A -85,B 0,C 180,E1 -5928.716,E2 -5928.716} C_VEL
LIN {X 0,Y 502.854,Z 135.845,A -85,B 0,C 180,E1 -5931.965,E2 -5931.965} C_VEL
LIN {X 0,Y 502.897,Z 135.846,A -85,B 0,C 180,E1 -5934.385,E2 -5934.385} C_VEL
LIN {X 0,Y 503.013,Z 135.823,A -85,B 0,C 180,E1 -5937.597,E2 -5937.597} C_VEL
LIN {X 0,Y 503.007,Z 135.829,A -85,B 0,C 180,E1 -5939.999,E2 -5939.999} C_VEL
LIN {X 0,Y 503.013,Z 135.828,A -85,B 0,C 180,E1 -5942.402,E2 -5942.402} C_VEL
LIN {X 0,Y 502.895,Z 135.84,A -85,B 0,C 180,E1 -5945.613,E2 -5945.613} C_VEL
LIN {X 0,Y 502.85,Z 135.852,A -85,B 0,C 180,E1 -5948.033,E2 -5948.033} C_VEL
LIN {X 0,Y 502.84,Z 135.845,A -85,B 0,C 180,E1 -5951.283,E2 -5951.283} C_VEL
LIN {X 0,Y 502.827,Z 135.847,A -85,B 0,C 180,E1 -5954.571,E2 -5954.571} C_VEL
LIN {X 0,Y 502.795,Z 135.854,A -85,B 0,C 180,E1 -5958.102,E2 -5958.102} C_VEL
LIN {X 0,Y 502.76,Z 135.857,A -85,B 0,C 180,E1 -5961.311,E2 -5961.311} C_VEL
LIN {X 0,Y 502.761,Z 135.859,A -85,B 0,C 180,E1 -5963.914,E2 -5963.914} C_VEL
LIN {X 0,Y 502.783,Z 135.851,A -85,B 0,C 180,E1 -5966.57,E2 -5966.57} C_VEL
LIN {X 0,Y 502.79,Z 135.853,A -85,B 0,C 180,E1 -5969.929,E2 -5969.929} C_VEL
LIN {X 0,Y 502.801,Z 135.852,A -85,B 0,C 180,E1 -5973.033,E2 -5973.033} C_VEL
LIN {X 0,Y 502.761,Z 135.855,A -85,B 0,C 180,E1 -5975.951,E2 -5975.951} C_VEL
LIN {X 0,Y 502.781,Z 135.856,A -85,B 0,C 180,E1 -5978.977,E2 -5978.977} C_VEL
LIN {X 0,Y 502.741,Z 135.856,A -85,B 0,C 180,E1 -5982.191,E2 -5982.191} C_VEL
LIN {X 0,Y 502.782,Z 135.855,A -85,B 0,C 180,E1 -5985.469,E2 -5985.469} C_VEL
LIN {X 0,Y 502.758,Z 135.861,A -85,B 0,C 180,E1 -5988.927,E2 -5988.927} C_VEL
LIN {X 0,Y 502.784,Z 135.851,A -85,B 0,C 180,E1 -5992.045,E2 -5992.045} C_VEL
LIN {X 0,Y 502.782,Z 135.858,A -85,B 0,C 180,E1 -5995.032,E2 -5995.032} C_VEL
LIN {X 0,Y 502.782,Z 135.855,A -85,B 0,C 180,E1 -5997.184,E2 -5997.184} C_VEL
LIN {X 0,Y 502.09,Z 135.939,A -85,B 0,C 180,E1 -5997.853,E2 -5997.853} C_VEL
LIN {X 0,Y 499.229,Z 136.301,A -85,B 0,C 180,E1 -5998.939,E2 -5998.939} C_VEL
LIN {X 0,Y 496.825,Z 136.597,A -85,B 0,C 180,E1 -5999.814,E2 -5999.814} C_VEL
LIN {X 0,Y 495.792,Z 136.727,A -85,B 0,C 180,E1 -6000.49,E2 -6000.49} C_VEL
LIN {X 0,Y 495.707,Z 136.733,A -85,B 0,C 180,E1 -6000.718,E2 -6000.718} C_VEL
LIN {X 0,Y 495.71,Z 136.733,A -85,B 0,C 180,E1 -6003.927,E2 -6003.927} C_VEL
LIN {X 0,Y 495.737,Z 136.731,A -85,B 0,C 180,E1 -6007.143,E2 -6007.143} C_VEL
LIN {X 0,Y 495.747,Z 136.731,A -85,B 0,C 180,E1 -6010.108,E2 -6010.108} C_VEL
LIN {X 0,Y 495.695,Z 136.74,A -85,B 0,C 180,E1 -6012.678,E2 -6012.678} C_VEL
LIN {X 0,Y 495.768,Z 136.725,A -85,B 0,C 180,E1 -6015.216,E2 -6015.216} C_VEL
LIN {X 0,Y 495.813,Z 136.725,A -85,B 0,C 180,E1 -6018.554,E2 -6018.554} C_VEL
LIN {X 0,Y 495.802,Z 136.724,A -85,B 0,C 180,E1 -6021.851,E2 -6021.851} C_VEL
LIN {X 0,Y 495.843,Z 136.723,A -85,B 0,C 180,E1 -6024.306,E2 -6024.306} C_VEL
LIN {X 0,Y 495.967,Z 136.704,A -85,B 0,C 180,E1 -6027.563,E2 -6027.563} C_VEL
LIN {X 0,Y 495.964,Z 136.71,A -85,B 0,C 180,E1 -6030,E2 -6030} C_VEL
LIN {X 0,Y 495.872,Z 136.742,A -85,B 0,C 180,E1 -6031.675,E2 -6031.675} C_VEL
LIN {X 0,Y 496.55,Z 142.412,A -85,B 0,C 180,E1 -6032.839,E2 -6032.839} C_VEL
LIN {X 0,Y 496.307,Z 157.817,A -85,B 0,C 180,E1 -6035.892,E2 -6035.892} C_VEL
LIN {X 0,Y 496.307,Z 158.46,A -85,B 0,C 180,E1 -6036.02,E2 -6036.02} C_VEL
LIN {X 0,Y 498.64,Z 171.109,A -85,B 0,C 180,E1 -6036.296,E2 -6036.296} C_VEL
LIN {X 0,Y 498.005,Z 265.176,A -85,B 0,C 180,E1 -6037.679,E2 -6037.679} C_VEL
LIN {X 0,Y 497.718,Z 278.614,A -85,B 0,C 180,E1 -6038.041,E2 -6038.041} C_VEL
LIN {X 0,Y 497.492,Z 291.386,A -85,B 0,C 180,E1 -6038.559,E2 -6038.559} C_VEL
LIN {X 0,Y 497.263,Z 302.183,A -85,B 0,C 180,E1 -6039.149,E2 -6039.149} C_VEL
LIN {X 0,Y 496.809,Z 314.026,A -85,B 0,C 180,E1 -6039.979,E2 -6039.979} C_VEL
LIN {X 0,Y 496.442,Z 324.611,A -85,B 0,C 180,E1 -6040.915,E2 -6040.915} C_VEL
LIN {X 0,Y 496.043,Z 334.443,A -85,B 0,C 180,E1 -6041.994,E2 -6041.994} C_VEL
LIN {X 0,Y 495.747,Z 342.653,A -85,B 0,C 180,E1 -6043.11,E2 -6043.11} C_VEL
LIN {X 0,Y 495.484,Z 350.182,A -85,B 0,C 180,E1 -6044.372,E2 -6044.372} C_VEL
LIN {X 0,Y 495.291,Z 356.216,A -85,B 0,C 180,E1 -6045.641,E2 -6045.641} C_VEL
LIN {X 0,Y 495.158,Z 360.951,A -85,B 0,C 180,E1 -6046.916,E2 -6046.916} C_VEL
LIN {X 0,Y 495.036,Z 364.532,A -85,B 0,C 180,E1 -6048.2,E2 -6048.2} C_VEL
LIN {X 0,Y 494.991,Z 366.297,A -85,B 0,C 180,E1 -6049.06,E2 -6049.06} C_VEL
LIN {X 0,Y 494.944,Z 368.181,A -85,B 0,C 180,E1 -6050.421,E2 -6050.421} C_VEL
LIN {X 0,Y 494.896,Z 368.93,A -85,B 0,C 180,E1 -6051.668,E2 -6051.668} C_VEL
LIN {X 0,Y 494.913,Z 368.893,A -85,B 0,C 180,E1 -6052.629,E2 -6052.629} C_VEL
LIN {X 0,Y 494.946,Z 368.429,A -85,B 0,C 180,E1 -6053.427,E2 -6053.427} C_VEL
LIN {X 0,Y 494.945,Z 366.959,A -85,B 0,C 180,E1 -6054.666,E2 -6054.666} C_VEL
LIN {X 0,Y 495.072,Z 364.018,A -85,B 0,C 180,E1 -6056.109,E2 -6056.109} C_VEL
LIN {X 0,Y 495.19,Z 359.99,A -85,B 0,C 180,E1 -6057.468,E2 -6057.468} C_VEL
LIN {X 0,Y 495.312,Z 354.542,A -85,B 0,C 180,E1 -6058.844,E2 -6058.844} C_VEL
LIN {X 0,Y 495.544,Z 348.15,A -85,B 0,C 180,E1 -6060.105,E2 -6060.105} C_VEL
LIN {X 0,Y 495.82,Z 339.89,A -85,B 0,C 180,E1 -6061.393,E2 -6061.393} C_VEL
LIN {X 0,Y 496.231,Z 330.573,A -85,B 0,C 180,E1 -6062.56,E2 -6062.56} C_VEL
LIN {X 0,Y 496.544,Z 321.308,A -85,B 0,C 180,E1 -6063.504,E2 -6063.504} C_VEL
LIN {X 0,Y 496.925,Z 311.332,A -85,B 0,C 180,E1 -6064.33,E2 -6064.33} C_VEL
LIN {X 0,Y 497.291,Z 299.173,A -85,B 0,C 180,E1 -6065.128,E2 -6065.128} C_VEL
LIN {X 0,Y 497.683,Z 286.643,A -85,B 0,C 180,E1 -6065.752,E2 -6065.752} C_VEL
LIN {X 0,Y 497.913,Z 274.436,A -85,B 0,C 180,E1 -6066.185,E2 -6066.185} C_VEL
LIN {X 0,Y 498.038,Z 261.799,A -85,B 0,C 180,E1 -6066.477,E2 -6066.477} C_VEL
LIN {X 0,Y 498.53,Z 169.789,A -85,B 0,C 180,E1 -6067.824,E2 -6067.824} C_VEL
LIN {X 0,Y 496.391,Z 158.544,A -85,B 0,C 180,E1 -6068.08,E2 -6068.08} C_VEL
LIN {X 0,Y 496.649,Z 143.532,A -85,B 0,C 180,E1 -6071.002,E2 -6071.002} C_VEL
LIN {X 0,Y 496.151,Z 138.718,A -85,B 0,C 180,E1 -6071.957,E2 -6071.957} C_VEL
LIN {X 0,Y 495.818,Z 136.728,A -85,B 0,C 180,E1 -6072.368,E2 -6072.368} C_VEL
LIN {X 0,Y 495.745,Z 136.732,A -85,B 0,C 180,E1 -6075.14,E2 -6075.14} C_VEL
LIN {X 0,Y 495.779,Z 136.73,A -85,B 0,C 180,E1 -6078.222,E2 -6078.222} C_VEL
LIN {X 0,Y 495.766,Z 136.729,A -85,B 0,C 180,E1 -6081.232,E2 -6081.232} C_VEL
LIN {X 0,Y 495.745,Z 136.73,A -85,B 0,C 180,E1 -6084.463,E2 -6084.463} C_VEL
LIN {X 0,Y 495.765,Z 136.733,A -85,B 0,C 180,E1 -6087.406,E2 -6087.406} C_VEL
LIN {X 0,Y 495.764,Z 136.726,A -85,B 0,C 180,E1 -6090.254,E2 -6090.254} C_VEL
LIN {X 0,Y 495.822,Z 136.726,A -85,B 0,C 180,E1 -6093.252,E2 -6093.252} C_VEL
LIN {X 0,Y 495.747,Z 136.731,A -85,B 0,C 180,E1 -6095.726,E2 -6095.726} C_VEL
LIN {X 0,Y 495.742,Z 136.73,A -85,B 0,C 180,E1 -6098.372,E2 -6098.372} C_VEL
LIN {X 0,Y 495.779,Z 136.732,A -85,B 0,C 180,E1 -6100.972,E2 -6100.972} C_VEL
LIN {X 0,Y 495.824,Z 136.722,A -85,B 0,C 180,E1 -6104.549,E2 -6104.549} C_VEL
LIN {X 0,Y 495.83,Z 136.718,A -85,B 0,C 180,E1 -6107.966,E2 -6107.966} C_VEL
LIN {X 0,Y 495.835,Z 136.719,A -85,B 0,C 180,E1 -6111.031,E2 -6111.031} C_VEL
LIN {X 0,Y 495.885,Z 136.715,A -85,B 0,C 180,E1 -6114.307,E2 -6114.307} C_VEL
LIN {X 0,Y 495.988,Z 136.697,A -85,B 0,C 180,E1 -6117.564,E2 -6117.564} C_VEL
LIN {X 0,Y 495.944,Z 136.703,A -85,B 0,C 180,E1 -6120.813,E2 -6120.813} C_VEL
LIN {X 0,Y 495.981,Z 136.705,A -85,B 0,C 180,E1 -6122.437,E2 -6122.437} C_VEL
LIN {X 0,Y 495.872,Z 136.71,A -85,B 0,C 180,E1 -6125.694,E2 -6125.694} C_VEL
LIN {X 0,Y 495.811,Z 136.719,A -85,B 0,C 180,E1 -6128.971,E2 -6128.971} C_VEL
LIN {X 0,Y 495.832,Z 136.721,A -85,B 0,C 180,E1 -6132.035,E2 -6132.035} C_VEL
LIN {X 0,Y 495.806,Z 136.722,A -85,B 0,C 180,E1 -6135.443,E2 -6135.443} C_VEL
LIN {X 0,Y 495.766,Z 136.727,A -85,B 0,C 180,E1 -6139.03,E2 -6139.03} C_VEL
LIN {X 0,Y 495.729,Z 136.734,A -85,B 0,C 180,E1 -6141.63,E2 -6141.63} C_VEL
LIN {X 0,Y 495.711,Z 136.734,A -85,B 0,C 180,E1 -6144.278,E2 -6144.278} C_VEL
LIN {X 0,Y 495.731,Z 136.729,A -85,B 0,C 180,E1 -6146.98,E2 -6146.98} C_VEL
LIN {X 0,Y 495.699,Z 136.732,A -85,B 0,C 180,E1 -6150.134,E2 -6150.134} C_VEL
LIN {X 0,Y 495.729,Z 136.738,A -85,B 0,C 180,E1 -6153.233,E2 -6153.233} C_VEL
LIN {X 0,Y 495.681,Z 136.737,A -85,B 0,C 180,E1 -6156.082,E2 -6156.082} C_VEL
LIN {X 0,Y 495.726,Z 136.733,A -85,B 0,C 180,E1 -6158.763,E2 -6158.763} C_VEL
LIN {X 0,Y 495.703,Z 136.736,A -85,B 0,C 180,E1 -6161.787,E2 -6161.787} C_VEL
LIN {X 0,Y 495.733,Z 136.738,A -85,B 0,C 180,E1 -6165.142,E2 -6165.142} C_VEL
LIN {X 0,Y 495.725,Z 136.735,A -85,B 0,C 180,E1 -6168.216,E2 -6168.216} C_VEL
LIN {X 0,Y 495.744,Z 136.732,A -85,B 0,C 180,E1 -6171.235,E2 -6171.235} C_VEL
LIN {X 0,Y 495.742,Z 136.734,A -85,B 0,C 180,E1 -6174.462,E2 -6174.462} C_VEL
LIN {X 0,Y 495.754,Z 136.729,A -85,B 0,C 180,E1 -6177.405,E2 -6177.405} C_VEL
LIN {X 0,Y 495.76,Z 136.733,A -85,B 0,C 180,E1 -6180.253,E2 -6180.253} C_VEL
LIN {X 0,Y 495.742,Z 136.733,A -85,B 0,C 180,E1 -6183.271,E2 -6183.271} C_VEL
LIN {X 0,Y 495.741,Z 136.781,A -85,B 0,C 180,E1 -6184.83,E2 -6184.83} C_VEL
LIN {X 0,Y 497.518,Z 146.241,A -85,B 0,C 180,E1 -6186.503,E2 -6186.503} C_VEL
LIN {X 0,Y 497.091,Z 161.734,A -85,B 0,C 180,E1 -6189.052,E2 -6189.052} C_VEL
LIN {X 0,Y 496.512,Z 180.346,A -85,B 0,C 180,E1 -6192.069,E2 -6192.069} C_VEL
LIN {X 0,Y 496.226,Z 192.082,A -85,B 0,C 180,E1 -6193.955,E2 -6193.955} C_VEL
LIN {X 0,Y 498.486,Z 207.957,A -85,B 0,C 180,E1 -6194.268,E2 -6194.268} C_VEL
LIN {X 0,Y 497.925,Z 301.237,A -85,B 0,C 180,E1 -6195.648,E2 -6195.648} C_VEL
LIN {X 0,Y 497.641,Z 314.286,A -85,B 0,C 180,E1 -6196.004,E2 -6196.004} C_VEL
LIN {X 0,Y 497.289,Z 326.911,A -85,B 0,C 180,E1 -6196.515,E2 -6196.515} C_VEL
LIN {X 0,Y 496.9,Z 338.298,A -85,B 0,C 180,E1 -6197.139,E2 -6197.139} C_VEL
LIN {X 0,Y 496.509,Z 349.798,A -85,B 0,C 180,E1 -6197.949,E2 -6197.949} C_VEL
LIN {X 0,Y 496.177,Z 360.292,A -85,B 0,C 180,E1 -6198.873,E2 -6198.873} C_VEL
LIN {X 0,Y 495.806,Z 368.87,A -85,B 0,C 180,E1 -6199.794,E2 -6199.794} C_VEL
LIN {X 0,Y 495.561,Z 376.79,A -85,B 0,C 180,E1 -6200.82,E2 -6200.82} C_VEL
LIN {X 0,Y 495.316,Z 384.525,A -85,B 0,C 180,E1 -6202.048,E2 -6202.048} C_VEL
LIN {X 0,Y 495.172,Z 389.825,A -85,B 0,C 180,E1 -6203.071,E2 -6203.071} C_VEL
LIN {X 0,Y 495.112,Z 394.964,A -85,B 0,C 180,E1 -6204.298,E2 -6204.298} C_VEL
LIN {X 0,Y 495.006,Z 398.951,A -85,B 0,C 180,E1 -6205.521,E2 -6205.521} C_VEL
LIN {X 0,Y 495.042,Z 401.902,A -85,B 0,C 180,E1 -6206.745,E2 -6206.745} C_VEL
LIN {X 0,Y 494.999,Z 403.305,A -85,B 0,C 180,E1 -6207.559,E2 -6207.559} C_VEL
LIN {X 0,Y 494.963,Z 404.307,A -85,B 0,C 180,E1 -6208.373,E2 -6208.373} C_VEL
LIN {X 0,Y 494.907,Z 405.139,A -85,B 0,C 180,E1 -6210,E2 -6210} C_VEL
LIN {X 0,Y 494.963,Z 404.321,A -85,B 0,C 180,E1 -6211.627,E2 -6211.627} C_VEL
LIN {X 0,Y 494.999,Z 403.326,A -85,B 0,C 180,E1 -6212.441,E2 -6212.441} C_VEL
LIN {X 0,Y 495.042,Z 401.929,A -85,B 0,C 180,E1 -6213.256,E2 -6213.256} C_VEL
LIN {X 0,Y 495.006,Z 398.985,A -85,B 0,C 180,E1 -6214.479,E2 -6214.479} C_VEL
LIN {X 0,Y 495.114,Z 395.003,A -85,B 0,C 180,E1 -6215.703,E2 -6215.703} C_VEL
LIN {X 0,Y 495.241,Z 388.873,A -85,B 0,C 180,E1 -6217.133,E2 -6217.133} C_VEL
LIN {X 0,Y 495.406,Z 382.176,A -85,B 0,C 180,E1 -6218.361,E2 -6218.361} C_VEL
LIN {X 0,Y 495.681,Z 373.868,A -85,B 0,C 180,E1 -6219.59,E2 -6219.59} C_VEL
LIN {X 0,Y 495.961,Z 365.345,A -85,B 0,C 180,E1 -6220.616,E2 -6220.616} C_VEL
LIN {X 0,Y 496.351,Z 354.818,A -85,B 0,C 180,E1 -6221.641,E2 -6221.641} C_VEL
LIN {X 0,Y 496.722,Z 343.268,A -85,B 0,C 180,E1 -6222.543,E2 -6222.543} C_VEL
LIN {X 0,Y 497.139,Z 331.026,A -85,B 0,C 180,E1 -6223.281,E2 -6223.281} C_VEL
LIN {X 0,Y 497.538,Z 318.604,A -85,B 0,C 180,E1 -6223.843,E2 -6223.843} C_VEL
LIN {X 0,Y 497.865,Z 305.792,A -85,B 0,C 180,E1 -6224.25,E2 -6224.25} C_VEL
LIN {X 0,Y 498.075,Z 292.213,A -85,B 0,C 180,E1 -6224.505,E2 -6224.505} C_VEL
LIN {X 0,Y 498.411,Z 206.974,A -85,B 0,C 180,E1 -6225.748,E2 -6225.748} C_VEL
LIN {X 0,Y 496.226,Z 192.344,A -85,B 0,C 180,E1 -6226.037,E2 -6226.037} C_VEL
LIN {X 0,Y 496.74,Z 174.079,A -85,B 0,C 180,E1 -6228.991,E2 -6228.991} C_VEL
LIN {X 0,Y 497.281,Z 158.38,A -85,B 0,C 180,E1 -6231.559,E2 -6231.559} C_VEL
LIN {X 0,Y 497.609,Z 146.724,A -85,B 0,C 180,E1 -6233.493,E2 -6233.493} C_VEL
LIN {X 0,Y 495.746,Z 136.733,A -85,B 0,C 180,E1 -6235.282,E2 -6235.282} C_VEL
LIN {X 0,Y 495.741,Z 136.73,A -85,B 0,C 180,E1 -6238.482,E2 -6238.482} C_VEL
LIN {X 0,Y 495.751,Z 136.73,A -85,B 0,C 180,E1 -6240.688,E2 -6240.688} C_VEL
LIN {X 0,Y 495.745,Z 136.737,A -85,B 0,C 180,E1 -6243.566,E2 -6243.566} C_VEL
LIN {X 0,Y 495.72,Z 136.731,A -85,B 0,C 180,E1 -6246.545,E2 -6246.545} C_VEL
LIN {X 0,Y 495.748,Z 136.733,A -85,B 0,C 180,E1 -6249.639,E2 -6249.639} C_VEL
LIN {X 0,Y 495.7,Z 136.736,A -85,B 0,C 180,E1 -6252.886,E2 -6252.886} C_VEL
LIN {X 0,Y 495.727,Z 136.731,A -85,B 0,C 180,E1 -6255.998,E2 -6255.998} C_VEL
LIN {X 0,Y 495.732,Z 136.737,A -85,B 0,C 180,E1 -6259.296,E2 -6259.296} C_VEL
LIN {X 0,Y 495.75,Z 136.732,A -85,B 0,C 180,E1 -6261.408,E2 -6261.408} C_VEL
LIN {X 0,Y 495.748,Z 136.729,A -85,B 0,C 180,E1 -6264.462,E2 -6264.462} C_VEL
LIN {X 0,Y 495.755,Z 136.73,A -85,B 0,C 180,E1 -6267.404,E2 -6267.404} C_VEL
LIN {X 0,Y 495.745,Z 136.729,A -85,B 0,C 180,E1 -6270.252,E2 -6270.252} C_VEL
LIN {X 0,Y 495.745,Z 136.731,A -85,B 0,C 180,E1 -6273.27,E2 -6273.27} C_VEL
LIN {X 0,Y 495.74,Z 136.735,A -85,B 0,C 180,E1 -6276.612,E2 -6276.612} C_VEL
LIN {X 0,Y 495.784,Z 136.724,A -85,B 0,C 180,E1 -6279.324,E2 -6279.324} C_VEL
LIN {X 0,Y 495.766,Z 136.726,A -85,B 0,C 180,E1 -6281.827,E2 -6281.827} C_VEL
LIN {X 0,Y 495.779,Z 136.725,A -85,B 0,C 180,E1 -6285.216,E2 -6285.216} C_VEL
LIN {X 0,Y 495.856,Z 136.722,A -85,B 0,C 180,E1 -6288.554,E2 -6288.554} C_VEL
LIN {X 0,Y 495.818,Z 136.721,A -85,B 0,C 180,E1 -6291.851,E2 -6291.851} C_VEL
LIN {X 0,Y 495.856,Z 136.722,A -85,B 0,C 180,E1 -6294.305,E2 -6294.305} C_VEL
LIN {X 0,Y 495.98,Z 136.699,A -85,B 0,C 180,E1 -6297.563,E2 -6297.563} C_VEL
LIN {X 0,Y 495.976,Z 136.705,A -85,B 0,C 180,E1 -6299.999,E2 -6299.999} C_VEL
LIN {X 0,Y 495.979,Z 136.704,A -85,B 0,C 180,E1 -6302.436,E2 -6302.436} C_VEL
LIN {X 0,Y 495.854,Z 136.718,A -85,B 0,C 180,E1 -6305.693,E2 -6305.693} C_VEL
LIN {X 0,Y 495.814,Z 136.726,A -85,B 0,C 180,E1 -6308.148,E2 -6308.148} C_VEL
LIN {X 0,Y 495.825,Z 136.72,A -85,B 0,C 180,E1 -6311.445,E2 -6311.445} C_VEL
LIN {X 0,Y 495.778,Z 136.724,A -85,B 0,C 180,E1 -6314.782,E2 -6314.782} C_VEL
LIN {X 0,Y 495.749,Z 136.73,A -85,B 0,C 180,E1 -6318.225,E2 -6318.225} C_VEL
LIN {X 0,Y 495.747,Z 136.728,A -85,B 0,C 180,E1 -6320.757,E2 -6320.757} C_VEL
LIN {X 0,Y 495.735,Z 136.734,A -85,B 0,C 180,E1 -6323.387,E2 -6323.387} C_VEL
LIN {X 0,Y 495.716,Z 136.734,A -85,B 0,C 180,E1 -6326.071,E2 -6326.071} C_VEL
LIN {X 0,Y 495.715,Z 136.732,A -85,B 0,C 180,E1 -6328.817,E2 -6328.817} C_VEL
LIN {X 0,Y 495.748,Z 136.732,A -85,B 0,C 180,E1 -6331.723,E2 -6331.723} C_VEL
LIN {X 0,Y 495.756,Z 136.727,A -85,B 0,C 180,E1 -6334.691,E2 -6334.691} C_VEL
LIN {X 0,Y 495.71,Z 136.737,A -85,B 0,C 180,E1 -6337.562,E2 -6337.562} C_VEL
LIN {X 0,Y 495.74,Z 136.729,A -85,B 0,C 180,E1 -6340.044,E2 -6340.044} C_VEL
LIN {X 0,Y 495.692,Z 136.739,A -85,B 0,C 180,E1 -6342.886,E2 -6342.886} C_VEL
LIN {X 0,Y 495.718,Z 136.731,A -85,B 0,C 180,E1 -6345.997,E2 -6345.997} C_VEL
LIN {X 0,Y 495.722,Z 136.736,A -85,B 0,C 180,E1 -6349.295,E2 -6349.295} C_VEL
LIN {X 0,Y 495.74,Z 136.732,A -85,B 0,C 180,E1 -6351.407,E2 -6351.407} C_VEL
LIN {X 0,Y 495.734,Z 136.732,A -85,B 0,C 180,E1 -6354.461,E2 -6354.461} C_VEL
LIN {X 0,Y 495.744,Z 136.73,A -85,B 0,C 180,E1 -6357.404,E2 -6357.404} C_VEL
LIN {X 0,Y 495.734,Z 136.731,A -85,B 0,C 180,E1 -6360.251,E2 -6360.251} C_VEL
LIN {X 0,Y 495.707,Z 136.733,A -85,B 0,C 180,E1 -6360.718,E2 -6360.718} C_VEL
LIN {X 0,Y 495.032,Z 136.82,A -85,B 0,C 180,E1 -6361.397,E2 -6361.397} C_VEL
LIN {X 0,Y 492.161,Z 137.18,A -85,B 0,C 180,E1 -6362.499,E2 -6362.499} C_VEL
LIN {X 0,Y 489.753,Z 137.476,A -85,B 0,C 180,E1 -6363.388,E2 -6363.388} C_VEL
LIN {X 0,Y 488.744,Z 137.602,A -85,B 0,C 180,E1 -6364.074,E2 -6364.074} C_VEL
LIN {X 0,Y 488.674,Z 137.612,A -85,B 0,C 180,E1 -6364.306,E2 -6364.306} C_VEL
LIN {X 0,Y 488.7,Z 137.607,A -85,B 0,C 180,E1 -6367.152,E2 -6367.152} C_VEL
LIN {X 0,Y 488.708,Z 137.605,A -85,B 0,C 180,E1 -6369.809,E2 -6369.809} C_VEL
LIN {X 0,Y 488.661,Z 137.618,A -85,B 0,C 180,E1 -6372.42,E2 -6372.42} C_VEL
LIN {X 0,Y 488.739,Z 137.602,A -85,B 0,C 180,E1 -6374.999,E2 -6374.999} C_VEL
LIN {X 0,Y 488.776,Z 137.604,A -85,B 0,C 180,E1 -6378.387,E2 -6378.387} C_VEL
LIN {X 0,Y 488.748,Z 137.602,A -85,B 0,C 180,E1 -6381.732,E2 -6381.732} C_VEL
LIN {X 0,Y 488.802,Z 137.601,A -85,B 0,C 180,E1 -6384.223,E2 -6384.223} C_VEL
LIN {X 0,Y 488.933,Z 137.581,A -85,B 0,C 180,E1 -6387.528,E2 -6387.528} C_VEL
LIN {X 0,Y 488.933,Z 137.585,A -85,B 0,C 180,E1 -6390,E2 -6390} C_VEL
LIN {X 0,Y 488.809,Z 137.714,A -85,B 0,C 180,E1 -6391.545,E2 -6391.545} C_VEL
LIN {X 0,Y 489.594,Z 144.12,A -85,B 0,C 180,E1 -6392.88,E2 -6392.88} C_VEL
LIN {X 0,Y 489.332,Z 158.733,A -85,B 0,C 180,E1 -6395.796,E2 -6395.796} C_VEL
LIN {X 0,Y 491.804,Z 171.461,A -85,B 0,C 180,E1 -6396.075,E2 -6396.075} C_VEL
LIN {X 0,Y 491.127,Z 265.451,A -85,B 0,C 180,E1 -6397.477,E2 -6397.477} C_VEL
LIN {X 0,Y 490.859,Z 278.84,A -85,B 0,C 180,E1 -6397.843,E2 -6397.843} C_VEL
LIN {X 0,Y 490.6,Z 291.834,A -85,B 0,C 180,E1 -6398.379,E2 -6398.379} C_VEL
LIN {X 0,Y 490.244,Z 304.084,A -85,B 0,C 180,E1 -6399.073,E2 -6399.073} C_VEL
LIN {X 0,Y 489.838,Z 315.579,A -85,B 0,C 180,E1 -6399.914,E2 -6399.914} C_VEL
LIN {X 0,Y 489.435,Z 325.941,A -85,B 0,C 180,E1 -6400.863,E2 -6400.863} C_VEL
LIN {X 0,Y 489.024,Z 334.984,A -85,B 0,C 180,E1 -6401.888,E2 -6401.888} C_VEL
LIN {X 0,Y 488.687,Z 343.615,A -85,B 0,C 180,E1 -6403.091,E2 -6403.091} C_VEL
LIN {X 0,Y 488.42,Z 351.021,A -85,B 0,C 180,E1 -6404.372,E2 -6404.372} C_VEL
LIN {X 0,Y 488.231,Z 356.484,A -85,B 0,C 180,E1 -6405.552,E2 -6405.552} C_VEL
LIN {X 0,Y 488.086,Z 360.859,A -85,B 0,C 180,E1 -6406.737,E2 -6406.737} C_VEL
LIN {X 0,Y 487.964,Z 364.668,A -85,B 0,C 180,E1 -6408.092,E2 -6408.092} C_VEL
LIN {X 0,Y 487.874,Z 367.135,A -85,B 0,C 180,E1 -6409.349,E2 -6409.349} C_VEL
LIN {X 0,Y 487.861,Z 368.588,A -85,B 0,C 180,E1 -6410.552,E2 -6410.552} C_VEL
LIN {X 0,Y 487.815,Z 369.254,A -85,B 0,C 180,E1 -6411.999,E2 -6411.999} C_VEL
LIN {X 0,Y 487.847,Z 369.035,A -85,B 0,C 180,E1 -6412.89,E2 -6412.89} C_VEL
LIN {X 0,Y 487.852,Z 368.362,A -85,B 0,C 180,E1 -6413.789,E2 -6413.789} C_VEL
LIN {X 0,Y 487.86,Z 367.003,A -85,B 0,C 180,E1 -6414.832,E2 -6414.832} C_VEL
LIN {X 0,Y 487.999,Z 364.563,A -85,B 0,C 180,E1 -6416.056,E2 -6416.056} C_VEL
LIN {X 0,Y 488.119,Z 360.634,A -85,B 0,C 180,E1 -6417.435,E2 -6417.435} C_VEL
LIN {X 0,Y 488.255,Z 354.967,A -85,B 0,C 180,E1 -6418.905,E2 -6418.905} C_VEL
LIN {X 0,Y 488.529,Z 347.798,A -85,B 0,C 180,E1 -6420.328,E2 -6420.328} C_VEL
LIN {X 0,Y 488.857,Z 339.287,A -85,B 0,C 180,E1 -6421.651,E2 -6421.651} C_VEL
LIN {X 0,Y 489.273,Z 329.745,A -85,B 0,C 180,E1 -6422.837,E2 -6422.837} C_VEL
LIN {X 0,Y 489.649,Z 320.211,A -85,B 0,C 180,E1 -6423.791,E2 -6423.791} C_VEL
LIN {X 0,Y 490.05,Z 309.905,A -85,B 0,C 180,E1 -6424.63,E2 -6424.63} C_VEL
LIN {X 0,Y 490.415,Z 299.103,A -85,B 0,C 180,E1 -6425.335,E2 -6425.335} C_VEL
LIN {X 0,Y 490.794,Z 286.823,A -85,B 0,C 180,E1 -6425.952,E2 -6425.952} C_VEL
LIN {X 0,Y 491.031,Z 274.017,A -85,B 0,C 180,E1 -6426.408,E2 -6426.408} C_VEL
LIN {X 0,Y 491.212,Z 260.884,A -85,B 0,C 180,E1 -6426.703,E2 -6426.703} C_VEL
LIN {X 0,Y 491.717,Z 170.791,A -85,B 0,C 180,E1 -6428.04,E2 -6428.04} C_VEL
LIN {X 0,Y 489.421,Z 158.884,A -85,B 0,C 180,E1 -6428.301,E2 -6428.301} C_VEL
LIN {X 0,Y 489.7,Z 144.733,A -85,B 0,C 180,E1 -6431.079,E2 -6431.079} C_VEL
LIN {X 0,Y 489.106,Z 139.448,A -85,B 0,C 180,E1 -6432.144,E2 -6432.144} C_VEL
LIN {X 0,Y 488.769,Z 137.605,A -85,B 0,C 180,E1 -6432.552,E2 -6432.552} C_VEL
LIN {X 0,Y 488.698,Z 137.615,A -85,B 0,C 180,E1 -6435.976,E2 -6435.976} C_VEL
LIN {X 0,Y 488.721,Z 137.607,A -85,B 0,C 180,E1 -6438.587,E2 -6438.587} C_VEL
LIN {X 0,Y 488.738,Z 137.603,A -85,B 0,C 180,E1 -6440.943,E2 -6440.943} C_VEL
LIN {X 0,Y 488.675,Z 137.616,A -85,B 0,C 180,E1 -6443.869,E2 -6443.869} C_VEL
LIN {X 0,Y 488.736,Z 137.603,A -85,B 0,C 180,E1 -6446.878,E2 -6446.878} C_VEL
LIN {X 0,Y 488.722,Z 137.607,A -85,B 0,C 180,E1 -6449.782,E2 -6449.782} C_VEL
LIN {X 0,Y 488.791,Z 137.6,A -85,B 0,C 180,E1 -6453.057,E2 -6453.057} C_VEL
LIN {X 0,Y 488.688,Z 137.608,A -85,B 0,C 180,E1 -6456.255,E2 -6456.255} C_VEL
LIN {X 0,Y 488.746,Z 137.606,A -85,B 0,C 180,E1 -6459.176,E2 -6459.176} C_VEL
LIN {X 0,Y 488.747,Z 137.602,A -85,B 0,C 180,E1 -6461.633,E2 -6461.633} C_VEL
LIN {X 0,Y 488.761,Z 137.605,A -85,B 0,C 180,E1 -6465,E2 -6465} C_VEL
LIN {X 0,Y 488.807,Z 137.595,A -85,B 0,C 180,E1 -6468.388,E2 -6468.388} C_VEL
LIN {X 0,Y 488.786,Z 137.593,A -85,B 0,C 180,E1 -6471.734,E2 -6471.734} C_VEL
LIN {X 0,Y 488.842,Z 137.591,A -85,B 0,C 180,E1 -6474.225,E2 -6474.225} C_VEL
LIN {X 0,Y 488.955,Z 137.573,A -85,B 0,C 180,E1 -6477.529,E2 -6477.529} C_VEL
LIN {X 0,Y 488.97,Z 137.573,A -85,B 0,C 180,E1 -6480.001,E2 -6480.001} C_VEL
LIN {X 0,Y 488.947,Z 137.581,A -85,B 0,C 180,E1 -6482.472,E2 -6482.472} C_VEL
LIN {X 0,Y 488.829,Z 137.588,A -85,B 0,C 180,E1 -6485.777,E2 -6485.777} C_VEL
LIN {X 0,Y 488.766,Z 137.604,A -85,B 0,C 180,E1 -6488.268,E2 -6488.268} C_VEL
LIN {X 0,Y 488.808,Z 137.589,A -85,B 0,C 180,E1 -6491.613,E2 -6491.613} C_VEL
LIN {X 0,Y 488.753,Z 137.599,A -85,B 0,C 180,E1 -6495.001,E2 -6495.001} C_VEL
LIN {X 0,Y 488.746,Z 137.602,A -85,B 0,C 180,E1 -6498.443,E2 -6498.443} C_VEL
LIN {X 0,Y 488.701,Z 137.605,A -85,B 0,C 180,E1 -6501.072,E2 -6501.072} C_VEL
LIN {X 0,Y 488.668,Z 137.617,A -85,B 0,C 180,E1 -6503.747,E2 -6503.747} C_VEL
LIN {X 0,Y 488.684,Z 137.605,A -85,B 0,C 180,E1 -6506.477,E2 -6506.477} C_VEL
LIN {X 0,Y 488.661,Z 137.617,A -85,B 0,C 180,E1 -6509.275,E2 -6509.275} C_VEL
LIN {X 0,Y 488.68,Z 137.609,A -85,B 0,C 180,E1 -6512.149,E2 -6512.149} C_VEL
LIN {X 0,Y 488.696,Z 137.61,A -85,B 0,C 180,E1 -6515.117,E2 -6515.117} C_VEL
LIN {X 0,Y 488.647,Z 137.611,A -85,B 0,C 180,E1 -6518.204,E2 -6518.204} C_VEL
LIN {X 0,Y 488.646,Z 137.618,A -85,B 0,C 180,E1 -6521.423,E2 -6521.423} C_VEL
LIN {X 0,Y 488.698,Z 137.614,A -85,B 0,C 180,E1 -6524.804,E2 -6524.804} C_VEL
LIN {X 0,Y 488.65,Z 137.617,A -85,B 0,C 180,E1 -6527.47,E2 -6527.47} C_VEL
LIN {X 0,Y 488.706,Z 137.608,A -85,B 0,C 180,E1 -6529.674,E2 -6529.674} C_VEL
LIN {X 0,Y 488.667,Z 137.613,A -85,B 0,C 180,E1 -6532.84,E2 -6532.84} C_VEL
LIN {X 0,Y 488.72,Z 137.605,A -85,B 0,C 180,E1 -6535.886,E2 -6535.886} C_VEL
LIN {X 0,Y 488.692,Z 137.613,A -85,B 0,C 180,E1 -6538.82,E2 -6538.82} C_VEL
LIN {X 0,Y 488.697,Z 137.61,A -85,B 0,C 180,E1 -6541.668,E2 -6541.668} C_VEL
LIN {X 0,Y 488.735,Z 137.757,A -85,B 0,C 180,E1 -6544.657,E2 -6544.657} C_VEL
LIN {X 0,Y 490.599,Z 147.84,A -85,B 0,C 180,E1 -6546.467,E2 -6546.467} C_VEL
LIN {X 0,Y 490.061,Z 164.308,A -85,B 0,C 180,E1 -6549.21,E2 -6549.21} C_VEL
LIN {X 0,Y 489.473,Z 182.716,A -85,B 0,C 180,E1 -6552.235,E2 -6552.235} C_VEL
LIN {X 0,Y 489.244,Z 191.858,A -85,B 0,C 180,E1 -6553.723,E2 -6553.723} C_VEL
LIN {X 0,Y 491.628,Z 209.2,A -85,B 0,C 180,E1 -6554.064,E2 -6554.064} C_VEL
LIN {X 0,Y 491.062,Z 300.986,A -85,B 0,C 180,E1 -6555.443,E2 -6555.443} C_VEL
LIN {X 0,Y 490.758,Z 314.028,A -85,B 0,C 180,E1 -6555.804,E2 -6555.804} C_VEL
LIN {X 0,Y 490.353,Z 326.648,A -85,B 0,C 180,E1 -6556.321,E2 -6556.321} C_VEL
LIN {X 0,Y 489.953,Z 337.882,A -85,B 0,C 180,E1 -6556.943,E2 -6556.943} C_VEL
LIN {X 0,Y 489.526,Z 349.531,A -85,B 0,C 180,E1 -6557.774,E2 -6557.774} C_VEL
LIN {X 0,Y 489.143,Z 360.023,A -85,B 0,C 180,E1 -6558.711,E2 -6558.711} C_VEL
LIN {X 0,Y 488.784,Z 368.602,A -85,B 0,C 180,E1 -6559.646,E2 -6559.646} C_VEL
LIN {X 0,Y 488.506,Z 376.521,A -85,B 0,C 180,E1 -6560.686,E2 -6560.686} C_VEL
LIN {X 0,Y 488.243,Z 384.257,A -85,B 0,C 180,E1 -6561.932,E2 -6561.932} C_VEL
LIN {X 0,Y 488.09,Z 389.558,A -85,B 0,C 180,E1 -6562.97,E2 -6562.97} C_VEL
LIN {X 0,Y 488.007,Z 394.699,A -85,B 0,C 180,E1 -6564.214,E2 -6564.214} C_VEL
LIN {X 0,Y 487.918,Z 398.689,A -85,B 0,C 180,E1 -6565.456,E2 -6565.456} C_VEL
LIN {X 0,Y 487.965,Z 401.641,A -85,B 0,C 180,E1 -6566.697,E2 -6566.697} C_VEL
LIN {X 0,Y 487.891,Z 404.048,A -85,B 0,C 180,E1 -6568.349,E2 -6568.349} C_VEL
LIN {X 0,Y 487.827,Z 404.881,A -85,B 0,C 180,E1 -6570,E2 -6570} C_VEL
LIN {X 0,Y 487.891,Z 404.062,A -85,B 0,C 180,E1 -6571.651,E2 -6571.651} C_VEL
LIN {X 0,Y 487.909,Z 403.067,A -85,B 0,C 180,E1 -6572.477,E2 -6572.477} C_VEL
LIN {X 0,Y 487.965,Z 401.67,A -85,B 0,C 180,E1 -6573.303,E2 -6573.303} C_VEL
LIN {X 0,Y 487.919,Z 398.725,A -85,B 0,C 180,E1 -6574.544,E2 -6574.544} C_VEL
LIN {X 0,Y 488.01,Z 394.741,A -85,B 0,C 180,E1 -6575.786,E2 -6575.786} C_VEL
LIN {X 0,Y 488.175,Z 388.609,A -85,B 0,C 180,E1 -6577.237,E2 -6577.237} C_VEL
LIN {X 0,Y 488.343,Z 381.909,A -85,B 0,C 180,E1 -6578.483,E2 -6578.483} C_VEL
LIN {X 0,Y 488.645,Z 373.599,A -85,B 0,C 180,E1 -6579.73,E2 -6579.73} C_VEL
LIN {X 0,Y 488.972,Z 365.072,A -85,B 0,C 180,E1 -6580.769,E2 -6580.769} C_VEL
LIN {X 0,Y 489.371,Z 354.537,A -85,B 0,C 180,E1 -6581.809,E2 -6581.809} C_VEL
LIN {X 0,Y 489.751,Z 343.052,A -85,B 0,C 180,E1 -6582.719,E2 -6582.719} C_VEL
LIN {X 0,Y 490.209,Z 330.721,A -85,B 0,C 180,E1 -6583.472,E2 -6583.472} C_VEL
LIN {X 0,Y 490.64,Z 318.281,A -85,B 0,C 180,E1 -6584.041,E2 -6584.041} C_VEL
LIN {X 0,Y 490.975,Z 305.429,A -85,B 0,C 180,E1 -6584.455,E2 -6584.455} C_VEL
LIN {X 0,Y 491.199,Z 289.991,A -85,B 0,C 180,E1 -6584.739,E2 -6584.739} C_VEL
LIN {X 0,Y 491.572,Z 207.765,A -85,B 0,C 180,E1 -6585.955,E2 -6585.955} C_VEL
LIN {X 0,Y 489.243,Z 192.084,A -85,B 0,C 180,E1 -6586.271,E2 -6586.271} C_VEL
LIN {X 0,Y 489.778,Z 173.817,A -85,B 0,C 180,E1 -6589.271,E2 -6589.271} C_VEL
LIN {X 0,Y 490.368,Z 158.126,A -85,B 0,C 180,E1 -6591.878,E2 -6591.878} C_VEL
LIN {X 0,Y 490.634,Z 147.639,A -85,B 0,C 180,E1 -6593.646,E2 -6593.646} C_VEL
LIN {X 0,Y 488.697,Z 137.609,A -85,B 0,C 180,E1 -6595.491,E2 -6595.491} C_VEL
LIN {X 0,Y 488.688,Z 137.608,A -85,B 0,C 180,E1 -6598.685,E2 -6598.685} C_VEL
LIN {X 0,Y 488.693,Z 137.612,A -85,B 0,C 180,E1 -6601.18,E2 -6601.18} C_VEL
LIN {X 0,Y 488.722,Z 137.605,A -85,B 0,C 180,E1 -6604.114,E2 -6604.114} C_VEL
LIN {X 0,Y 488.674,Z 137.613,A -85,B 0,C 180,E1 -6607.16,E2 -6607.16} C_VEL
LIN {X 0,Y 488.698,Z 137.606,A -85,B 0,C 180,E1 -6610.341,E2 -6610.341} C_VEL
LIN {X 0,Y 488.678,Z 137.613,A -85,B 0,C 180,E1 -6613.656,E2 -6613.656} C_VEL
LIN {X 0,Y 488.678,Z 137.608,A -85,B 0,C 180,E1 -6616.344,E2 -6616.344} C_VEL
LIN {X 0,Y 488.708,Z 137.607,A -85,B 0,C 180,E1 -6619.673,E2 -6619.673} C_VEL
LIN {X 0,Y 488.675,Z 137.613,A -85,B 0,C 180,E1 -6622.84,E2 -6622.84} C_VEL
LIN {X 0,Y 488.723,Z 137.603,A -85,B 0,C 180,E1 -6625.886,E2 -6625.886} C_VEL
LIN {X 0,Y 488.687,Z 137.614,A -85,B 0,C 180,E1 -6628.819,E2 -6628.819} C_VEL
LIN {X 0,Y 488.698,Z 137.606,A -85,B 0,C 180,E1 -6631.668,E2 -6631.668} C_VEL
LIN {X 0,Y 488.695,Z 137.609,A -85,B 0,C 180,E1 -6634.441,E2 -6634.441} C_VEL
LIN {X 0,Y 488.712,Z 137.607,A -85,B 0,C 180,E1 -6637.152,E2 -6637.152} C_VEL
LIN {X 0,Y 488.721,Z 137.603,A -85,B 0,C 180,E1 -6639.81,E2 -6639.81} C_VEL
LIN {X 0,Y 488.675,Z 137.614,A -85,B 0,C 180,E1 -6642.421,E2 -6642.421} C_VEL
LIN {X 0,Y 488.751,Z 137.602,A -85,B 0,C 180,E1 -6644.999,E2 -6644.999} C_VEL
LIN {X 0,Y 488.811,Z 137.599,A -85,B 0,C 180,E1 -6648.387,E2 -6648.387} C_VEL
LIN {X 0,Y 488.765,Z 137.598,A -85,B 0,C 180,E1 -6651.732,E2 -6651.732} C_VEL
LIN {X 0,Y 488.816,Z 137.598,A -85,B 0,C 180,E1 -6654.223,E2 -6654.223} C_VEL
LIN {X 0,Y 488.946,Z 137.576,A -85,B 0,C 180,E1 -6657.528,E2 -6657.528} C_VEL
LIN {X 0,Y 488.945,Z 137.58,A -85,B 0,C 180,E1 -6659.999,E2 -6659.999} C_VEL
LIN {X 0,Y 488.945,Z 137.579,A -85,B 0,C 180,E1 -6662.471,E2 -6662.471} C_VEL
LIN {X 0,Y 488.814,Z 137.596,A -85,B 0,C 180,E1 -6665.776,E2 -6665.776} C_VEL
LIN {X 0,Y 488.76,Z 137.603,A -85,B 0,C 180,E1 -6668.267,E2 -6668.267} C_VEL
LIN {X 0,Y 488.787,Z 137.599,A -85,B 0,C 180,E1 -6671.612,E2 -6671.612} C_VEL
LIN {X 0,Y 488.744,Z 137.6,A -85,B 0,C 180,E1 -6675,E2 -6675} C_VEL
LIN {X 0,Y 488.707,Z 137.606,A -85,B 0,C 180,E1 -6678.443,E2 -6678.443} C_VEL
LIN {X 0,Y 488.691,Z 137.608,A -85,B 0,C 180,E1 -6681.071,E2 -6681.071} C_VEL
LIN {X 0,Y 488.666,Z 137.617,A -85,B 0,C 180,E1 -6683.746,E2 -6683.746} C_VEL
LIN {X 0,Y 488.681,Z 137.608,A -85,B 0,C 180,E1 -6686.475,E2 -6686.475} C_VEL
LIN {X 0,Y 488.686,Z 137.612,A -85,B 0,C 180,E1 -6689.272,E2 -6689.272} C_VEL
LIN {X 0,Y 488.694,Z 137.607,A -85,B 0,C 180,E1 -6692.147,E2 -6692.147} C_VEL
LIN {X 0,Y 488.709,Z 137.609,A -85,B 0,C 180,E1 -6695.115,E2 -6695.115} C_VEL
LIN {X 0,Y 488.659,Z 137.611,A -85,B 0,C 180,E1 -6698.201,E2 -6698.201} C_VEL
LIN {X 0,Y 488.691,Z 137.607,A -85,B 0,C 180,E1 -6700.34,E2 -6700.34} C_VEL
LIN {X 0,Y 488.67,Z 137.612,A -85,B 0,C 180,E1 -6703.655,E2 -6703.655} C_VEL
LIN {X 0,Y 488.669,Z 137.61,A -85,B 0,C 180,E1 -6706.343,E2 -6706.343} C_VEL
LIN {X 0,Y 488.699,Z 137.607,A -85,B 0,C 180,E1 -6709.673,E2 -6709.673} C_VEL
LIN {X 0,Y 488.663,Z 137.617,A -85,B 0,C 180,E1 -6712.839,E2 -6712.839} C_VEL
LIN {X 0,Y 488.712,Z 137.604,A -85,B 0,C 180,E1 -6715.885,E2 -6715.885} C_VEL
LIN {X 0,Y 488.677,Z 137.617,A -85,B 0,C 180,E1 -6718.819,E2 -6718.819} C_VEL
LIN {X 0,Y 488.686,Z 137.607,A -85,B 0,C 180,E1 -6721.667,E2 -6721.667} C_VEL
LIN {X 0,Y 488.674,Z 137.612,A -85,B 0,C 180,E1 -6724.306,E2 -6724.306} C_VEL
LIN {X 0,Y 488.04,Z 137.696,A -85,B 0,C 180,E1 -6724.994,E2 -6724.994} C_VEL
LIN {X 0,Y 485.191,Z 138.049,A -85,B 0,C 180,E1 -6726.111,E2 -6726.111} C_VEL
LIN {X 0,Y 482.758,Z 138.349,A -85,B 0,C 180,E1 -6727.011,E2 -6727.011} C_VEL
LIN {X 0,Y 481.706,Z 138.477,A -85,B 0,C 180,E1 -6727.707,E2 -6727.707} C_VEL
LIN {X 0,Y 481.618,Z 138.489,A -85,B 0,C 180,E1 -6727.943,E2 -6727.943} C_VEL
LIN {X 0,Y 481.685,Z 138.486,A -85,B 0,C 180,E1 -6730.392,E2 -6730.392} C_VEL
LIN {X 0,Y 481.606,Z 138.491,A -85,B 0,C 180,E1 -6733.031,E2 -6733.031} C_VEL
LIN {X 0,Y 481.665,Z 138.482,A -85,B 0,C 180,E1 -6735.638,E2 -6735.638} C_VEL
LIN {X 0,Y 481.727,Z 138.481,A -85,B 0,C 180,E1 -6738.214,E2 -6738.214} C_VEL
LIN {X 0,Y 481.707,Z 138.478,A -85,B 0,C 180,E1 -6741.611,E2 -6741.611} C_VEL
LIN {X 0,Y 481.764,Z 138.477,A -85,B 0,C 180,E1 -6744.139,E2 -6744.139} C_VEL
LIN {X 0,Y 481.899,Z 138.457,A -85,B 0,C 180,E1 -6747.492,E2 -6747.492} C_VEL
LIN {X 0,Y 481.902,Z 138.461,A -85,B 0,C 180,E1 -6750,E2 -6750} C_VEL
LIN {X 0,Y 481.753,Z 138.587,A -85,B 0,C 180,E1 -6751.384,E2 -6751.384} C_VEL
LIN {X 0,Y 482.617,Z 144.877,A -85,B 0,C 180,E1 -6752.713,E2 -6752.713} C_VEL
LIN {X 0,Y 482.382,Z 159.196,A -85,B 0,C 180,E1 -6755.565,E2 -6755.565} C_VEL
LIN {X 0,Y 484.907,Z 171.995,A -85,B 0,C 180,E1 -6755.849,E2 -6755.849} C_VEL
LIN {X 0,Y 484.269,Z 265.68,A -85,B 0,C 180,E1 -6757.269,E2 -6757.269} C_VEL
LIN {X 0,Y 483.989,Z 279.078,A -85,B 0,C 180,E1 -6757.64,E2 -6757.64} C_VEL
LIN {X 0,Y 483.709,Z 292.349,A -85,B 0,C 180,E1 -6758.196,E2 -6758.196} C_VEL
LIN {X 0,Y 483.381,Z 303.769,A -85,B 0,C 180,E1 -6758.85,E2 -6758.85} C_VEL
LIN {X 0,Y 482.966,Z 314.523,A -85,B 0,C 180,E1 -6759.633,E2 -6759.633} C_VEL
LIN {X 0,Y 482.52,Z 325.129,A -85,B 0,C 180,E1 -6760.596,E2 -6760.596} C_VEL
LIN {X 0,Y 482.143,Z 333.797,A -85,B 0,C 180,E1 -6761.562,E2 -6761.562} C_VEL
LIN {X 0,Y 481.754,Z 341.794,A -85,B 0,C 180,E1 -6762.64,E2 -6762.64} C_VEL
LIN {X 0,Y 481.435,Z 349.567,A -85,B 0,C 180,E1 -6763.938,E2 -6763.938} C_VEL
LIN {X 0,Y 481.212,Z 355.808,A -85,B 0,C 180,E1 -6765.241,E2 -6765.241} C_VEL
LIN {X 0,Y 481.043,Z 360.746,A -85,B 0,C 180,E1 -6766.552,E2 -6766.552} C_VEL
LIN {X 0,Y 480.899,Z 364.518,A -85,B 0,C 180,E1 -6767.872,E2 -6767.872} C_VEL
LIN {X 0,Y 480.827,Z 366.438,A -85,B 0,C 180,E1 -6768.757,E2 -6768.757} C_VEL
LIN {X 0,Y 480.764,Z 367.859,A -85,B 0,C 180,E1 -6769.647,E2 -6769.647} C_VEL
LIN {X 0,Y 480.758,Z 368.984,A -85,B 0,C 180,E1 -6770.679,E2 -6770.679} C_VEL
LIN {X 0,Y 480.74,Z 369.468,A -85,B 0,C 180,E1 -6772.34,E2 -6772.34} C_VEL
LIN {X 0,Y 480.756,Z 369.101,A -85,B 0,C 180,E1 -6773.247,E2 -6773.247} C_VEL
LIN {X 0,Y 480.755,Z 368.26,A -85,B 0,C 180,E1 -6774.162,E2 -6774.162} C_VEL
LIN {X 0,Y 480.796,Z 366.908,A -85,B 0,C 180,E1 -6775.081,E2 -6775.081} C_VEL
LIN {X 0,Y 480.938,Z 363.94,A -85,B 0,C 180,E1 -6776.468,E2 -6776.468} C_VEL
LIN {X 0,Y 481.116,Z 359.706,A -85,B 0,C 180,E1 -6777.869,E2 -6777.869} C_VEL
LIN {X 0,Y 481.287,Z 353.985,A -85,B 0,C 180,E1 -6779.287,E2 -6779.287} C_VEL
LIN {X 0,Y 481.569,Z 346.517,A -85,B 0,C 180,E1 -6780.716,E2 -6780.716} C_VEL
LIN {X 0,Y 481.862,Z 339.024,A -85,B 0,C 180,E1 -6781.868,E2 -6781.868} C_VEL
LIN {X 0,Y 482.303,Z 329.978,A -85,B 0,C 180,E1 -6782.999,E2 -6782.999} C_VEL
LIN {X 0,Y 482.719,Z 320.148,A -85,B 0,C 180,E1 -6783.993,E2 -6783.993} C_VEL
LIN {X 0,Y 483.221,Z 308.511,A -85,B 0,C 180,E1 -6784.937,E2 -6784.937} C_VEL
LIN {X 0,Y 483.651,Z 296.96,A -85,B 0,C 180,E1 -6785.666,E2 -6785.666} C_VEL
LIN {X 0,Y 483.996,Z 284.03,A -85,B 0,C 180,E1 -6786.279,E2 -6786.279} C_VEL
LIN {X 0,Y 484.227,Z 271.273,A -85,B 0,C 180,E1 -6786.704,E2 -6786.704} C_VEL
LIN {X 0,Y 484.401,Z 257.757,A -85,B 0,C 180,E1 -6786.969,E2 -6786.969} C_VEL
LIN {X 0,Y 484.932,Z 171.744,A -85,B 0,C 180,E1 -6788.262,E2 -6788.262} C_VEL
LIN {X 0,Y 482.469,Z 159.082,A -85,B 0,C 180,E1 -6788.555,E2 -6788.555} C_VEL
LIN {X 0,Y 482.738,Z 145.795,A -85,B 0,C 180,E1 -6791.185,E2 -6791.185} C_VEL
LIN {X 0,Y 482.042,Z 140.107,A -85,B 0,C 180,E1 -6792.352,E2 -6792.352} C_VEL
LIN {X 0,Y 481.71,Z 138.484,A -85,B 0,C 180,E1 -6792.713,E2 -6792.713} C_VEL
LIN {X 0,Y 481.655,Z 138.489,A -85,B 0,C 180,E1 -6795.641,E2 -6795.641} C_VEL
LIN {X 0,Y 481.67,Z 138.488,A -85,B 0,C 180,E1 -6798.085,E2 -6798.085} C_VEL
LIN {X 0,Y 481.694,Z 138.482,A -85,B 0,C 180,E1 -6801.144,E2 -6801.144} C_VEL
LIN {X 0,Y 481.659,Z 138.485,A -85,B 0,C 180,E1 -6804.797,E2 -6804.797} C_VEL
LIN {X 0,Y 481.669,Z 138.488,A -85,B 0,C 180,E1 -6807.327,E2 -6807.327} C_VEL
LIN {X 0,Y 481.677,Z 138.48,A -85,B 0,C 180,E1 -6810.26,E2 -6810.26} C_VEL
LIN {X 0,Y 481.744,Z 138.478,A -85,B 0,C 180,E1 -6813.113,E2 -6813.113} C_VEL
LIN {X 0,Y 481.673,Z 138.483,A -85,B 0,C 180,E1 -6815.888,E2 -6815.888} C_VEL
LIN {X 0,Y 481.702,Z 138.484,A -85,B 0,C 180,E1 -6819.028,E2 -6819.028} C_VEL
LIN {X 0,Y 481.688,Z 138.479,A -85,B 0,C 180,E1 -6822.159,E2 -6822.159} C_VEL
LIN {X 0,Y 481.742,Z 138.479,A -85,B 0,C 180,E1 -6824.777,E2 -6824.777} C_VEL
LIN {X 0,Y 481.752,Z 138.472,A -85,B 0,C 180,E1 -6828.216,E2 -6828.216} C_VEL
LIN {X 0,Y 481.741,Z 138.47,A -85,B 0,C 180,E1 -6831.612,E2 -6831.612} C_VEL
LIN {X 0,Y 481.801,Z 138.467,A -85,B 0,C 180,E1 -6834.14,E2 -6834.14} C_VEL
LIN {X 0,Y 481.922,Z 138.449,A -85,B 0,C 180,E1 -6837.493,E2 -6837.493} C_VEL
LIN {X 0,Y 481.941,Z 138.448,A -85,B 0,C 180,E1 -6840.001,E2 -6840.001} C_VEL
LIN {X 0,Y 481.912,Z 138.456,A -85,B 0,C 180,E1 -6842.508,E2 -6842.508} C_VEL
LIN {X 0,Y 481.788,Z 138.466,A -85,B 0,C 180,E1 -6845.861,E2 -6845.861} C_VEL
LIN {X 0,Y 481.725,Z 138.479,A -85,B 0,C 180,E1 -6848.39,E2 -6848.39} C_VEL
LIN {X 0,Y 481.754,Z 138.47,A -85,B 0,C 180,E1 -6851.785,E2 -6851.785} C_VEL
LIN {X 0,Y 481.734,Z 138.474,A -85,B 0,C 180,E1 -6855.225,E2 -6855.225} C_VEL
LIN {X 0,Y 481.706,Z 138.478,A -85,B 0,C 180,E1 -6858.723,E2 -6858.723} C_VEL
LIN {X 0,Y 481.637,Z 138.488,A -85,B 0,C 180,E1 -6861.396,E2 -6861.396} C_VEL
LIN {X 0,Y 481.648,Z 138.487,A -85,B 0,C 180,E1 -6864.115,E2 -6864.115} C_VEL
LIN {X 0,Y 481.653,Z 138.484,A -85,B 0,C 180,E1 -6867.117,E2 -6867.117} C_VEL
LIN {X 0,Y 481.602,Z 138.491,A -85,B 0,C 180,E1 -6869.747,E2 -6869.747} C_VEL
LIN {X 0,Y 481.635,Z 138.488,A -85,B 0,C 180,E1 -6872.678,E2 -6872.678} C_VEL
LIN {X 0,Y 481.641,Z 138.49,A -85,B 0,C 180,E1 -6875.2,E2 -6875.2} C_VEL
LIN {X 0,Y 481.623,Z 138.486,A -85,B 0,C 180,E1 -6878.002,E2 -6878.002} C_VEL
LIN {X 0,Y 481.606,Z 138.496,A -85,B 0,C 180,E1 -6881.048,E2 -6881.048} C_VEL
LIN {X 0,Y 481.652,Z 138.487,A -85,B 0,C 180,E1 -6884.459,E2 -6884.459} C_VEL
LIN {X 0,Y 481.614,Z 138.497,A -85,B 0,C 180,E1 -6886.856,E2 -6886.856} C_VEL
LIN {X 0,Y 481.658,Z 138.487,A -85,B 0,C 180,E1 -6890.058,E2 -6890.058} C_VEL
LIN {X 0,Y 481.622,Z 138.487,A -85,B 0,C 180,E1 -6893.378,E2 -6893.378} C_VEL
LIN {X 0,Y 481.673,Z 138.486,A -85,B 0,C 180,E1 -6896.327,E2 -6896.327} C_VEL
LIN {X 0,Y 481.648,Z 138.487,A -85,B 0,C 180,E1 -6899.419,E2 -6899.419} C_VEL
LIN {X 0,Y 481.653,Z 138.491,A -85,B 0,C 180,E1 -6902.165,E2 -6902.165} C_VEL
LIN {X 0,Y 481.696,Z 138.502,A -85,B 0,C 180,E1 -6904.434,E2 -6904.434} C_VEL
LIN {X 0,Y 483.608,Z 148.622,A -85,B 0,C 180,E1 -6906.284,E2 -6906.284} C_VEL
LIN {X 0,Y 483.283,Z 160.099,A -85,B 0,C 180,E1 -6908.234,E2 -6908.234} C_VEL
LIN {X 0,Y 482.636,Z 178.52,A -85,B 0,C 180,E1 -6911.316,E2 -6911.316} C_VEL
LIN {X 0,Y 482.24,Z 191.545,A -85,B 0,C 180,E1 -6913.473,E2 -6913.473} C_VEL
LIN {X 0,Y 484.801,Z 209.109,A -85,B 0,C 180,E1 -6913.834,E2 -6913.834} C_VEL
LIN {X 0,Y 484.21,Z 300.764,A -85,B 0,C 180,E1 -6915.232,E2 -6915.232} C_VEL
LIN {X 0,Y 483.873,Z 313.785,A -85,B 0,C 180,E1 -6915.598,E2 -6915.598} C_VEL
LIN {X 0,Y 483.443,Z 326.395,A -85,B 0,C 180,E1 -6916.121,E2 -6916.121} C_VEL
LIN {X 0,Y 482.994,Z 337.936,A -85,B 0,C 180,E1 -6916.773,E2 -6916.773} C_VEL
LIN {X 0,Y 482.555,Z 349.374,A -85,B 0,C 180,E1 -6917.604,E2 -6917.604} C_VEL
LIN {X 0,Y 482.157,Z 359.76,A -85,B 0,C 180,E1 -6918.545,E2 -6918.545} C_VEL
LIN {X 0,Y 481.775,Z 368.34,A -85,B 0,C 180,E1 -6919.494,E2 -6919.494} C_VEL
LIN {X 0,Y 481.454,Z 376.258,A -85,B 0,C 180,E1 -6920.548,E2 -6920.548} C_VEL
LIN {X 0,Y 481.172,Z 383.995,A -85,B 0,C 180,E1 -6921.813,E2 -6921.813} C_VEL
LIN {X 0,Y 481.017,Z 389.297,A -85,B 0,C 180,E1 -6922.866,E2 -6922.866} C_VEL
LIN {X 0,Y 480.91,Z 394.437,A -85,B 0,C 180,E1 -6924.129,E2 -6924.129} C_VEL
LIN {X 0,Y 480.837,Z 398.428,A -85,B 0,C 180,E1 -6925.389,E2 -6925.389} C_VEL
LIN {X 0,Y 480.888,Z 401.382,A -85,B 0,C 180,E1 -6926.649,E2 -6926.649} C_VEL
LIN {X 0,Y 480.822,Z 403.79,A -85,B 0,C 180,E1 -6928.325,E2 -6928.325} C_VEL
LIN {X 0,Y 480.751,Z 404.622,A -85,B 0,C 180,E1 -6930,E2 -6930} C_VEL
LIN {X 0,Y 480.822,Z 403.804,A -85,B 0,C 180,E1 -6931.675,E2 -6931.675} C_VEL
LIN {X 0,Y 480.889,Z 401.41,A -85,B 0,C 180,E1 -6933.352,E2 -6933.352} C_VEL
LIN {X 0,Y 480.837,Z 398.463,A -85,B 0,C 180,E1 -6934.611,E2 -6934.611} C_VEL
LIN {X 0,Y 480.915,Z 394.476,A -85,B 0,C 180,E1 -6935.872,E2 -6935.872} C_VEL
LIN {X 0,Y 481.103,Z 388.342,A -85,B 0,C 180,E1 -6937.344,E2 -6937.344} C_VEL
LIN {X 0,Y 481.298,Z 381.638,A -85,B 0,C 180,E1 -6938.608,E2 -6938.608} C_VEL
LIN {X 0,Y 481.583,Z 373.321,A -85,B 0,C 180,E1 -6939.874,E2 -6939.874} C_VEL
LIN {X 0,Y 481.965,Z 364.789,A -85,B 0,C 180,E1 -6940.928,E2 -6940.928} C_VEL
LIN {X 0,Y 482.392,Z 354.373,A -85,B 0,C 180,E1 -6941.971,E2 -6941.971} C_VEL
LIN {X 0,Y 482.812,Z 342.528,A -85,B 0,C 180,E1 -6942.922,E2 -6942.922} C_VEL
LIN {X 0,Y 483.293,Z 330.407,A -85,B 0,C 180,E1 -6943.669,E2 -6943.669} C_VEL
LIN {X 0,Y 483.765,Z 317.951,A -85,B 0,C 180,E1 -6944.245,E2 -6944.245} C_VEL
LIN {X 0,Y 484.114,Z 305.054,A -85,B 0,C 180,E1 -6944.664,E2 -6944.664} C_VEL
LIN {X 0,Y 484.321,Z 289.535,A -85,B 0,C 180,E1 -6944.953,E2 -6944.953} C_VEL
LIN {X 0,Y 484.728,Z 208.476,A -85,B 0,C 180,E1 -6946.169,E2 -6946.169} C_VEL
LIN {X 0,Y 482.248,Z 191.833,A -85,B 0,C 180,E1 -6946.511,E2 -6946.511} C_VEL
LIN {X 0,Y 482.793,Z 174.809,A -85,B 0,C 180,E1 -6949.349,E2 -6949.349} C_VEL
LIN {X 0,Y 483.479,Z 157.858,A -85,B 0,C 180,E1 -6952.207,E2 -6952.207} C_VEL
LIN {X 0,Y 483.697,Z 148.908,A -85,B 0,C 180,E1 -6953.74,E2 -6953.74} C_VEL
LIN {X 0,Y 481.687,Z 138.482,A -85,B 0,C 180,E1 -6955.674,E2 -6955.674} C_VEL
LIN {X 0,Y 481.643,Z 138.486,A -85,B 0,C 180,E1 -6958.895,E2 -6958.895} C_VEL
LIN {X 0,Y 481.654,Z 138.486,A -85,B 0,C 180,E1 -6962.188,E2 -6962.188} C_VEL
LIN {X 0,Y 481.662,Z 138.486,A -85,B 0,C 180,E1 -6965.203,E2 -6965.203} C_VEL
LIN {X 0,Y 481.67,Z 138.483,A -85,B 0,C 180,E1 -6968.86,E2 -6968.86} C_VEL
LIN {X 0,Y 481.62,Z 138.488,A -85,B 0,C 180,E1 -6972.164,E2 -6972.164} C_VEL
LIN {X 0,Y 481.658,Z 138.483,A -85,B 0,C 180,E1 -6974.458,E2 -6974.458} C_VEL
LIN {X 0,Y 481.62,Z 138.491,A -85,B 0,C 180,E1 -6976.855,E2 -6976.855} C_VEL
LIN {X 0,Y 481.662,Z 138.483,A -85,B 0,C 180,E1 -6980.057,E2 -6980.057} C_VEL
LIN {X 0,Y 481.625,Z 138.493,A -85,B 0,C 180,E1 -6983.252,E2 -6983.252} C_VEL
LIN {X 0,Y 481.675,Z 138.481,A -85,B 0,C 180,E1 -6986.327,E2 -6986.327} C_VEL
LIN {X 0,Y 481.639,Z 138.488,A -85,B 0,C 180,E1 -6989.421,E2 -6989.421} C_VEL
LIN {X 0,Y 481.655,Z 138.484,A -85,B 0,C 180,E1 -6992.165,E2 -6992.165} C_VEL
LIN {X 0,Y 481.678,Z 138.487,A -85,B 0,C 180,E1 -6994.967,E2 -6994.967} C_VEL
LIN {X 0,Y 481.641,Z 138.485,A -85,B 0,C 180,E1 -6997.704,E2 -6997.704} C_VEL
LIN {X 0,Y 481.698,Z 138.482,A -85,B 0,C 180,E1 -7000.392,E2 -7000.392} C_VEL
LIN {X 0,Y 481.619,Z 138.491,A -85,B 0,C 180,E1 -7003.031,E2 -7003.031} C_VEL
LIN {X 0,Y 481.676,Z 138.481,A -85,B 0,C 180,E1 -7005.638,E2 -7005.638} C_VEL
LIN {X 0,Y 481.756,Z 138.475,A -85,B 0,C 180,E1 -7008.215,E2 -7008.215} C_VEL
LIN {X 0,Y 481.723,Z 138.475,A -85,B 0,C 180,E1 -7011.61,E2 -7011.61} C_VEL
LIN {X 0,Y 481.777,Z 138.473,A -85,B 0,C 180,E1 -7014.138,E2 -7014.138} C_VEL
LIN {X 0,Y 481.911,Z 138.452,A -85,B 0,C 180,E1 -7017.492,E2 -7017.492} C_VEL
LIN {X 0,Y 481.914,Z 138.456,A -85,B 0,C 180,E1 -7019.999,E2 -7019.999} C_VEL
LIN {X 0,Y 481.91,Z 138.455,A -85,B 0,C 180,E1 -7022.507,E2 -7022.507} C_VEL
LIN {X 0,Y 481.776,Z 138.473,A -85,B 0,C 180,E1 -7025.86,E2 -7025.86} C_VEL
LIN {X 0,Y 481.719,Z 138.479,A -85,B 0,C 180,E1 -7028.388,E2 -7028.388} C_VEL
LIN {X 0,Y 481.738,Z 138.479,A -85,B 0,C 180,E1 -7031.784,E2 -7031.784} C_VEL
LIN {X 0,Y 481.724,Z 138.476,A -85,B 0,C 180,E1 -7035.224,E2 -7035.224} C_VEL
LIN {X 0,Y 481.651,Z 138.484,A -85,B 0,C 180,E1 -7038.723,E2 -7038.723} C_VEL
LIN {X 0,Y 481.63,Z 138.49,A -85,B 0,C 180,E1 -7041.395,E2 -7041.395} C_VEL
LIN {X 0,Y 481.646,Z 138.487,A -85,B 0,C 180,E1 -7044.114,E2 -7044.114} C_VEL
LIN {X 0,Y 481.651,Z 138.486,A -85,B 0,C 180,E1 -7047.116,E2 -7047.116} C_VEL
LIN {X 0,Y 481.652,Z 138.489,A -85,B 0,C 180,E1 -7049.742,E2 -7049.742} C_VEL
LIN {X 0,Y 481.65,Z 138.484,A -85,B 0,C 180,E1 -7052.675,E2 -7052.675} C_VEL
LIN {X 0,Y 481.626,Z 138.491,A -85,B 0,C 180,E1 -7055.709,E2 -7055.709} C_VEL
LIN {X 0,Y 481.631,Z 138.489,A -85,B 0,C 180,E1 -7058.862,E2 -7058.862} C_VEL
LIN {X 0,Y 481.617,Z 138.489,A -85,B 0,C 180,E1 -7061.907,E2 -7061.907} C_VEL
LIN {X 0,Y 481.65,Z 138.485,A -85,B 0,C 180,E1 -7064.457,E2 -7064.457} C_VEL
LIN {X 0,Y 481.611,Z 138.494,A -85,B 0,C 180,E1 -7066.854,E2 -7066.854} C_VEL
LIN {X 0,Y 481.652,Z 138.484,A -85,B 0,C 180,E1 -7070.057,E2 -7070.057} C_VEL
LIN {X 0,Y 481.613,Z 138.493,A -85,B 0,C 180,E1 -7073.251,E2 -7073.251} C_VEL
LIN {X 0,Y 481.665,Z 138.484,A -85,B 0,C 180,E1 -7076.326,E2 -7076.326} C_VEL
LIN {X 0,Y 481.628,Z 138.488,A -85,B 0,C 180,E1 -7079.42,E2 -7079.42} C_VEL
LIN {X 0,Y 481.643,Z 138.486,A -85,B 0,C 180,E1 -7082.164,E2 -7082.164} C_VEL
LIN {X 0,Y 481.666,Z 138.486,A -85,B 0,C 180,E1 -7084.967,E2 -7084.967} C_VEL
LIN {X 0,Y 481.618,Z 138.489,A -85,B 0,C 180,E1 -7087.943,E2 -7087.943} C_VEL
LIN {X 0,Y 480.956,Z 138.578,A -85,B 0,C 180,E1 -7088.641,E2 -7088.641} C_VEL
LIN {X 0,Y 478.142,Z 138.923,A -85,B 0,C 180,E1 -7089.775,E2 -7089.775} C_VEL
LIN {X 0,Y 475.756,Z 139.224,A -85,B 0,C 180,E1 -7090.689,E2 -7090.689} C_VEL
LIN {X 0,Y 474.721,Z 139.348,A -85,B 0,C 180,E1 -7091.395,E2 -7091.395} C_VEL
LIN {X 0,Y 474.63,Z 139.358,A -85,B 0,C 180,E1 -7091.634,E2 -7091.634} C_VEL
LIN {X 0,Y 474.68,Z 139.359,A -85,B 0,C 180,E1 -7094.543,E2 -7094.543} C_VEL
LIN {X 0,Y 474.685,Z 139.356,A -85,B 0,C 180,E1 -7098.037,E2 -7098.037} C_VEL
LIN {X 0,Y 474.656,Z 139.356,A -85,B 0,C 180,E1 -7101.485,E2 -7101.485} C_VEL
LIN {X 0,Y 474.727,Z 139.353,A -85,B 0,C 180,E1 -7104.052,E2 -7104.052} C_VEL
LIN {X 0,Y 474.864,Z 139.333,A -85,B 0,C 180,E1 -7107.455,E2 -7107.455} C_VEL
LIN {X 0,Y 474.871,Z 139.337,A -85,B 0,C 180,E1 -7110,E2 -7110} C_VEL
LIN {X 0,Y 474.702,Z 139.48,A -85,B 0,C 180,E1 -7111.219,E2 -7111.219} C_VEL
LIN {X 0,Y 475.635,Z 145.631,A -85,B 0,C 180,E1 -7112.54,E2 -7112.54} C_VEL
LIN {X 0,Y 475.393,Z 159.136,A -85,B 0,C 180,E1 -7115.301,E2 -7115.301} C_VEL
LIN {X 0,Y 478.169,Z 173.715,A -85,B 0,C 180,E1 -7115.641,E2 -7115.641} C_VEL
LIN {X 0,Y 477.411,Z 265.884,A -85,B 0,C 180,E1 -7117.055,E2 -7117.055} C_VEL
LIN {X 0,Y 477.107,Z 279.313,A -85,B 0,C 180,E1 -7117.432,E2 -7117.432} C_VEL
LIN {X 0,Y 476.837,Z 292.564,A -85,B 0,C 180,E1 -7117.995,E2 -7117.995} C_VEL
LIN {X 0,Y 476.485,Z 303.475,A -85,B 0,C 180,E1 -7118.623,E2 -7118.623} C_VEL
LIN {X 0,Y 476.044,Z 314.759,A -85,B 0,C 180,E1 -7119.453,E2 -7119.453} C_VEL
LIN {X 0,Y 475.58,Z 325.367,A -85,B 0,C 180,E1 -7120.429,E2 -7120.429} C_VEL
LIN {X 0,Y 475.085,Z 334.936,A -85,B 0,C 180,E1 -7121.52,E2 -7121.52} C_VEL
LIN {X 0,Y 474.669,Z 344.128,A -85,B 0,C 180,E1 -7122.832,E2 -7122.832} C_VEL
LIN {X 0,Y 474.335,Z 351.543,A -85,B 0,C 180,E1 -7124.151,E2 -7124.151} C_VEL
LIN {X 0,Y 474.099,Z 357.607,A -85,B 0,C 180,E1 -7125.52,E2 -7125.52} C_VEL
LIN {X 0,Y 473.926,Z 362.061,A -85,B 0,C 180,E1 -7126.808,E2 -7126.808} C_VEL
LIN {X 0,Y 473.775,Z 365.886,A -85,B 0,C 180,E1 -7128.312,E2 -7128.312} C_VEL
LIN {X 0,Y 473.682,Z 368.564,A -85,B 0,C 180,E1 -7129.953,E2 -7129.953} C_VEL
LIN {X 0,Y 473.647,Z 369.366,A -85,B 0,C 180,E1 -7130.862,E2 -7130.862} C_VEL
LIN {X 0,Y 473.617,Z 369.73,A -85,B 0,C 180,E1 -7131.776,E2 -7131.776} C_VEL
LIN {X 0,Y 473.66,Z 369.462,A -85,B 0,C 180,E1 -7133.086,E2 -7133.086} C_VEL
LIN {X 0,Y 473.695,Z 368.062,A -85,B 0,C 180,E1 -7134.546,E2 -7134.546} C_VEL
LIN {X 0,Y 473.822,Z 365.588,A -85,B 0,C 180,E1 -7135.948,E2 -7135.948} C_VEL
LIN {X 0,Y 473.972,Z 361.904,A -85,B 0,C 180,E1 -7137.365,E2 -7137.365} C_VEL
LIN {X 0,Y 474.094,Z 357.355,A -85,B 0,C 180,E1 -7138.667,E2 -7138.667} C_VEL
LIN {X 0,Y 474.354,Z 351.359,A -85,B 0,C 180,E1 -7140.002,E2 -7140.002} C_VEL
LIN {X 0,Y 474.636,Z 344.583,A -85,B 0,C 180,E1 -7141.215,E2 -7141.215} C_VEL
LIN {X 0,Y 475.093,Z 335.509,A -85,B 0,C 180,E1 -7142.523,E2 -7142.523} C_VEL
LIN {X 0,Y 475.554,Z 325.7,A -85,B 0,C 180,E1 -7143.655,E2 -7143.655} C_VEL
LIN {X 0,Y 475.969,Z 315.635,A -85,B 0,C 180,E1 -7144.593,E2 -7144.593} C_VEL
LIN {X 0,Y 476.52,Z 304.036,A -85,B 0,C 180,E1 -7145.454,E2 -7145.454} C_VEL
LIN {X 0,Y 476.923,Z 292.559,A -85,B 0,C 180,E1 -7146.118,E2 -7146.118} C_VEL
LIN {X 0,Y 477.192,Z 279.657,A -85,B 0,C 180,E1 -7146.667,E2 -7146.667} C_VEL
LIN {X 0,Y 477.431,Z 267.225,A -85,B 0,C 180,E1 -7147.025,E2 -7147.025} C_VEL
LIN {X 0,Y 478.124,Z 185.899,A -85,B 0,C 180,E1 -7148.287,E2 -7148.287} C_VEL
LIN {X 0,Y 478.156,Z 172.601,A -85,B 0,C 180,E1 -7148.493,E2 -7148.493} C_VEL
LIN {X 0,Y 475.507,Z 159.222,A -85,B 0,C 180,E1 -7148.826,E2 -7148.826} C_VEL
LIN {X 0,Y 475.796,Z 146.65,A -85,B 0,C 180,E1 -7151.341,E2 -7151.341} C_VEL
LIN {X 0,Y 474.693,Z 139.357,A -85,B 0,C 180,E1 -7152.893,E2 -7152.893} C_VEL
LIN {X 0,Y 474.631,Z 139.36,A -85,B 0,C 180,E1 -7156.515,E2 -7156.515} C_VEL
LIN {X 0,Y 474.637,Z 139.364,A -85,B 0,C 180,E1 -7159.345,E2 -7159.345} C_VEL
LIN {X 0,Y 474.613,Z 139.37,A -85,B 0,C 180,E1 -7161.704,E2 -7161.704} C_VEL
LIN {X 0,Y 474.622,Z 139.362,A -85,B 0,C 180,E1 -7164.726,E2 -7164.726} C_VEL
LIN {X 0,Y 474.633,Z 139.363,A -85,B 0,C 180,E1 -7167.789,E2 -7167.789} C_VEL
LIN {X 0,Y 474.622,Z 139.361,A -85,B 0,C 180,E1 -7170.885,E2 -7170.885} C_VEL
LIN {X 0,Y 474.66,Z 139.362,A -85,B 0,C 180,E1 -7173.629,E2 -7173.629} C_VEL
LIN {X 0,Y 474.635,Z 139.36,A -85,B 0,C 180,E1 -7176.642,E2 -7176.642} C_VEL
LIN {X 0,Y 474.653,Z 139.357,A -85,B 0,C 180,E1 -7180.09,E2 -7180.09} C_VEL
LIN {X 0,Y 474.635,Z 139.362,A -85,B 0,C 180,E1 -7182.775,E2 -7182.775} C_VEL
LIN {X 0,Y 474.646,Z 139.358,A -85,B 0,C 180,E1 -7185.422,E2 -7185.422} C_VEL
LIN {X 0,Y 474.705,Z 139.349,A -85,B 0,C 180,E1 -7188.038,E2 -7188.038} C_VEL
LIN {X 0,Y 474.712,Z 139.346,A -85,B 0,C 180,E1 -7191.487,E2 -7191.487} C_VEL
LIN {X 0,Y 474.747,Z 139.344,A -85,B 0,C 180,E1 -7194.905,E2 -7194.905} C_VEL
LIN {X 0,Y 474.887,Z 139.325,A -85,B 0,C 180,E1 -7197.456,E2 -7197.456} C_VEL
LIN {X 0,Y 474.911,Z 139.324,A -85,B 0,C 180,E1 -7200.001,E2 -7200.001} C_VEL
LIN {X 0,Y 474.877,Z 139.332,A -85,B 0,C 180,E1 -7202.545,E2 -7202.545} C_VEL
LIN {X 0,Y 474.749,Z 139.343,A -85,B 0,C 180,E1 -7205.949,E2 -7205.949} C_VEL
LIN {X 0,Y 474.7,Z 139.352,A -85,B 0,C 180,E1 -7208.515,E2 -7208.515} C_VEL
LIN {X 0,Y 474.707,Z 139.35,A -85,B 0,C 180,E1 -7211.963,E2 -7211.963} C_VEL
LIN {X 0,Y 474.692,Z 139.353,A -85,B 0,C 180,E1 -7215.457,E2 -7215.457} C_VEL
LIN {X 0,Y 474.66,Z 139.356,A -85,B 0,C 180,E1 -7219.011,E2 -7219.011} C_VEL
LIN {X 0,Y 474.58,Z 139.367,A -85,B 0,C 180,E1 -7221.73,E2 -7221.73} C_VEL
LIN {X 0,Y 474.627,Z 139.359,A -85,B 0,C 180,E1 -7224.495,E2 -7224.495} C_VEL
LIN {X 0,Y 474.599,Z 139.365,A -85,B 0,C 180,E1 -7227.327,E2 -7227.327} C_VEL
LIN {X 0,Y 474.551,Z 139.366,A -85,B 0,C 180,E1 -7230.235,E2 -7230.235} C_VEL
LIN {X 0,Y 474.61,Z 139.369,A -85,B 0,C 180,E1 -7233.223,E2 -7233.223} C_VEL
LIN {X 0,Y 474.567,Z 139.368,A -85,B 0,C 180,E1 -7236.326,E2 -7236.326} C_VEL
LIN {X 0,Y 474.599,Z 139.367,A -85,B 0,C 180,E1 -7239.551,E2 -7239.551} C_VEL
LIN {X 0,Y 474.568,Z 139.376,A -85,B 0,C 180,E1 -7242.94,E2 -7242.94} C_VEL
LIN {X 0,Y 474.582,Z 139.368,A -85,B 0,C 180,E1 -7245.892,E2 -7245.892} C_VEL
LIN {X 0,Y 474.601,Z 139.37,A -85,B 0,C 180,E1 -7249.045,E2 -7249.045} C_VEL
LIN {X 0,Y 474.597,Z 139.365,A -85,B 0,C 180,E1 -7251.707,E2 -7251.707} C_VEL
LIN {X 0,Y 474.62,Z 139.367,A -85,B 0,C 180,E1 -7254.725,E2 -7254.725} C_VEL
LIN {X 0,Y 474.63,Z 139.362,A -85,B 0,C 180,E1 -7257.787,E2 -7257.787} C_VEL
LIN {X 0,Y 474.601,Z 139.368,A -85,B 0,C 180,E1 -7260.891,E2 -7260.891} C_VEL
LIN {X 0,Y 474.642,Z 139.393,A -85,B 0,C 180,E1 -7264.23,E2 -7264.23} C_VEL
LIN {X 0,Y 476.694,Z 150.269,A -85,B 0,C 180,E1 -7266.249,E2 -7266.249} C_VEL
LIN {X 0,Y 476.255,Z 163.417,A -85,B 0,C 180,E1 -7268.511,E2 -7268.511} C_VEL
LIN {X 0,Y 475.496,Z 183.517,A -85,B 0,C 180,E1 -7271.917,E2 -7271.917} C_VEL
LIN {X 0,Y 475.252,Z 191.269,A -85,B 0,C 180,E1 -7273.219,E2 -7273.219} C_VEL
LIN {X 0,Y 477.976,Z 209.992,A -85,B 0,C 180,E1 -7273.611,E2 -7273.611} C_VEL
LIN {X 0,Y 477.363,Z 300.566,A -85,B 0,C 180,E1 -7275.015,E2 -7275.015} C_VEL
LIN {X 0,Y 477.056,Z 312.801,A -85,B 0,C 180,E1 -7275.36,E2 -7275.36} C_VEL
LIN {X 0,Y 476.585,Z 325.03,A -85,B 0,C 180,E1 -7275.863,E2 -7275.863} C_VEL
LIN {X 0,Y 476.082,Z 337.378,A -85,B 0,C 180,E1 -7276.556,E2 -7276.556} C_VEL
LIN {X 0,Y 475.633,Z 348.603,A -85,B 0,C 180,E1 -7277.377,E2 -7277.377} C_VEL
LIN {X 0,Y 475.18,Z 359.507,A -85,B 0,C 180,E1 -7278.374,E2 -7278.374} C_VEL
LIN {X 0,Y 474.746,Z 368.083,A -85,B 0,C 180,E1 -7279.336,E2 -7279.336} C_VEL
LIN {X 0,Y 474.425,Z 376,A -85,B 0,C 180,E1 -7280.407,E2 -7280.407} C_VEL
LIN {X 0,Y 474.129,Z 383.736,A -85,B 0,C 180,E1 -7281.69,E2 -7281.69} C_VEL
LIN {X 0,Y 473.897,Z 390.867,A -85,B 0,C 180,E1 -7283.186,E2 -7283.186} C_VEL
LIN {X 0,Y 473.836,Z 395.618,A -85,B 0,C 180,E1 -7284.468,E2 -7284.468} C_VEL
LIN {X 0,Y 473.734,Z 399.246,A -85,B 0,C 180,E1 -7285.746,E2 -7285.746} C_VEL
LIN {X 0,Y 473.795,Z 401.123,A -85,B 0,C 180,E1 -7286.599,E2 -7286.599} C_VEL
LIN {X 0,Y 473.725,Z 403.531,A -85,B 0,C 180,E1 -7288.3,E2 -7288.3} C_VEL
LIN {X 0,Y 473.693,Z 404.144,A -85,B 0,C 180,E1 -7289.15,E2 -7289.15} C_VEL
LIN {X 0,Y 473.677,Z 404.364,A -85,B 0,C 180,E1 -7290,E2 -7290} C_VEL
LIN {X 0,Y 473.693,Z 404.15,A -85,B 0,C 180,E1 -7290.85,E2 -7290.85} C_VEL
LIN {X 0,Y 473.725,Z 403.544,A -85,B 0,C 180,E1 -7291.7,E2 -7291.7} C_VEL
LIN {X 0,Y 473.742,Z 402.547,A -85,B 0,C 180,E1 -7292.551,E2 -7292.551} C_VEL
LIN {X 0,Y 473.796,Z 401.148,A -85,B 0,C 180,E1 -7293.402,E2 -7293.402} C_VEL
LIN {X 0,Y 473.76,Z 398.2,A -85,B 0,C 180,E1 -7294.68,E2 -7294.68} C_VEL
LIN {X 0,Y 473.823,Z 394.21,A -85,B 0,C 180,E1 -7295.96,E2 -7295.96} C_VEL
LIN {X 0,Y 474.013,Z 388.071,A -85,B 0,C 180,E1 -7297.454,E2 -7297.454} C_VEL
LIN {X 0,Y 474.245,Z 381.364,A -85,B 0,C 180,E1 -7298.737,E2 -7298.737} C_VEL
LIN {X 0,Y 474.541,Z 373.042,A -85,B 0,C 180,E1 -7300.022,E2 -7300.022} C_VEL
LIN {X 0,Y 474.944,Z 364.502,A -85,B 0,C 180,E1 -7301.091,E2 -7301.091} C_VEL
LIN {X 0,Y 475.399,Z 354.28,A -85,B 0,C 180,E1 -7302.131,E2 -7302.131} C_VEL
LIN {X 0,Y 475.8,Z 343.505,A -85,B 0,C 180,E1 -7303.018,E2 -7303.018} C_VEL
LIN {X 0,Y 476.314,Z 332.042,A -85,B 0,C 180,E1 -7303.764,E2 -7303.764} C_VEL
LIN {X 0,Y 476.783,Z 320.198,A -85,B 0,C 180,E1 -7304.349,E2 -7304.349} C_VEL
LIN {X 0,Y 477.196,Z 306.533,A -85,B 0,C 180,E1 -7304.827,E2 -7304.827} C_VEL
LIN {X 0,Y 477.443,Z 294.293,A -85,B 0,C 180,E1 -7305.092,E2 -7305.092} C_VEL
LIN {X 0,Y 477.92,Z 209.237,A -85,B 0,C 180,E1 -7306.387,E2 -7306.387} C_VEL
LIN {X 0,Y 475.266,Z 191.565,A -85,B 0,C 180,E1 -7306.76,E2 -7306.76} C_VEL
LIN {X 0,Y 475.805,Z 174.718,A -85,B 0,C 180,E1 -7309.613,E2 -7309.613} C_VEL
LIN {X 0,Y 476.463,Z 160.212,A -85,B 0,C 180,E1 -7312.094,E2 -7312.094} C_VEL
LIN {X 0,Y 476.779,Z 150.492,A -85,B 0,C 180,E1 -7313.781,E2 -7313.781} C_VEL
LIN {X 0,Y 474.625,Z 139.362,A -85,B 0,C 180,E1 -7315.901,E2 -7315.901} C_VEL
LIN {X 0,Y 474.604,Z 139.367,A -85,B 0,C 180,E1 -7319.253,E2 -7319.253} C_VEL
LIN {X 0,Y 474.606,Z 139.362,A -85,B 0,C 180,E1 -7322.428,E2 -7322.428} C_VEL
LIN {X 0,Y 474.614,Z 139.368,A -85,B 0,C 180,E1 -7325.468,E2 -7325.468} C_VEL
LIN {X 0,Y 474.612,Z 139.361,A -85,B 0,C 180,E1 -7328.458,E2 -7328.458} C_VEL
LIN {X 0,Y 474.597,Z 139.366,A -85,B 0,C 180,E1 -7331.789,E2 -7331.789} C_VEL
LIN {X 0,Y 474.621,Z 139.361,A -85,B 0,C 180,E1 -7334.702,E2 -7334.702} C_VEL
LIN {X 0,Y 474.581,Z 139.366,A -85,B 0,C 180,E1 -7337.77,E2 -7337.77} C_VEL
LIN {X 0,Y 474.626,Z 139.359,A -85,B 0,C 180,E1 -7340.452,E2 -7340.452} C_VEL
LIN {X 0,Y 474.589,Z 139.365,A -85,B 0,C 180,E1 -7343.676,E2 -7343.676} C_VEL
LIN {X 0,Y 474.619,Z 139.365,A -85,B 0,C 180,E1 -7346.777,E2 -7346.777} C_VEL
LIN {X 0,Y 474.59,Z 139.364,A -85,B 0,C 180,E1 -7349.768,E2 -7349.768} C_VEL
LIN {X 0,Y 474.643,Z 139.362,A -85,B 0,C 180,E1 -7352.676,E2 -7352.676} C_VEL
LIN {X 0,Y 474.63,Z 139.359,A -85,B 0,C 180,E1 -7355.505,E2 -7355.505} C_VEL
LIN {X 0,Y 474.629,Z 139.365,A -85,B 0,C 180,E1 -7358.887,E2 -7358.887} C_VEL
LIN {X 0,Y 474.635,Z 139.358,A -85,B 0,C 180,E1 -7361.883,E2 -7361.883} C_VEL
LIN {X 0,Y 474.693,Z 139.358,A -85,B 0,C 180,E1 -7364.543,E2 -7364.543} C_VEL
LIN {X 0,Y 474.71,Z 139.351,A -85,B 0,C 180,E1 -7368.037,E2 -7368.037} C_VEL
LIN {X 0,Y 474.672,Z 139.353,A -85,B 0,C 180,E1 -7371.485,E2 -7371.485} C_VEL
LIN {X 0,Y 474.741,Z 139.349,A -85,B 0,C 180,E1 -7374.051,E2 -7374.051} C_VEL
LIN {X 0,Y 474.876,Z 139.328,A -85,B 0,C 180,E1 -7377.455,E2 -7377.455} C_VEL
LIN {X 0,Y 474.884,Z 139.332,A -85,B 0,C 180,E1 -7379.999,E2 -7379.999} C_VEL
LIN {X 0,Y 474.875,Z 139.331,A -85,B 0,C 180,E1 -7382.544,E2 -7382.544} C_VEL
LIN {X 0,Y 474.739,Z 139.351,A -85,B 0,C 180,E1 -7385.947,E2 -7385.947} C_VEL
LIN {X 0,Y 474.668,Z 139.356,A -85,B 0,C 180,E1 -7388.514,E2 -7388.514} C_VEL
LIN {X 0,Y 474.696,Z 139.358,A -85,B 0,C 180,E1 -7391.962,E2 -7391.962} C_VEL
LIN {X 0,Y 474.683,Z 139.355,A -85,B 0,C 180,E1 -7395.455,E2 -7395.455} C_VEL
LIN {X 0,Y 474.605,Z 139.362,A -85,B 0,C 180,E1 -7399.012,E2 -7399.012} C_VEL
LIN {X 0,Y 474.576,Z 139.373,A -85,B 0,C 180,E1 -7401.729,E2 -7401.729} C_VEL
LIN {X 0,Y 474.625,Z 139.359,A -85,B 0,C 180,E1 -7404.494,E2 -7404.494} C_VEL
LIN {X 0,Y 474.597,Z 139.367,A -85,B 0,C 180,E1 -7407.325,E2 -7407.325} C_VEL
LIN {X 0,Y 474.584,Z 139.365,A -85,B 0,C 180,E1 -7410.231,E2 -7410.231} C_VEL
LIN {X 0,Y 474.613,Z 139.366,A -85,B 0,C 180,E1 -7413.221,E2 -7413.221} C_VEL
LIN {X 0,Y 474.58,Z 139.365,A -85,B 0,C 180,E1 -7416.323,E2 -7416.323} C_VEL
LIN {X 0,Y 474.598,Z 139.366,A -85,B 0,C 180,E1 -7419.643,E2 -7419.643} C_VEL
LIN {X 0,Y 474.566,Z 139.371,A -85,B 0,C 180,E1 -7422.939,E2 -7422.939} C_VEL
LIN {X 0,Y 474.598,Z 139.363,A -85,B 0,C 180,E1 -7425.893,E2 -7425.893} C_VEL
LIN {X 0,Y 474.586,Z 139.368,A -85,B 0,C 180,E1 -7429.338,E2 -7429.338} C_VEL
LIN {X 0,Y 474.601,Z 139.363,A -85,B 0,C 180,E1 -7431.704,E2 -7431.704} C_VEL
LIN {X 0,Y 474.612,Z 139.366,A -85,B 0,C 180,E1 -7434.724,E2 -7434.724} C_VEL
LIN {X 0,Y 474.62,Z 139.36,A -85,B 0,C 180,E1 -7437.786,E2 -7437.786} C_VEL
LIN {X 0,Y 474.587,Z 139.37,A -85,B 0,C 180,E1 -7440.891,E2 -7440.891} C_VEL
